LIN {X 0,Y 457.681,Z 997.987,A -85,B 0,C 180,E1 -8390.375,E2 -8390.375} C_VEL
LIN {X 0,Y 458.676,Z 987.154,A -85,B 0,C 180,E1 -8391.458,E2 -8391.458} C_VEL
LIN {X 0,Y 459.714,Z 975.478,A -85,B 0,C 180,E1 -8392.469,E2 -8392.469} C_VEL
LIN {X 0,Y 460.765,Z 963.447,A -85,B 0,C 180,E1 -8393.364,E2 -8393.364} C_VEL
LIN {X 0,Y 461.763,Z 951.373,A -85,B 0,C 180,E1 -8394.128,E2 -8394.128} C_VEL
LIN {X 0,Y 462.621,Z 938.572,A -85,B 0,C 180,E1 -8394.813,E2 -8394.813} C_VEL
LIN {X 0,Y 463.49,Z 925.141,A -85,B 0,C 180,E1 -8395.393,E2 -8395.393} C_VEL
LIN {X 0,Y 464.076,Z 912.216,A -85,B 0,C 180,E1 -8395.84,E2 -8395.84} C_VEL
LIN {X 0,Y 464.663,Z 898.95,A -85,B 0,C 180,E1 -8396.175,E2 -8396.175} C_VEL
LIN {X 0,Y 465.199,Z 876.109,A -85,B 0,C 180,E1 -8396.57,E2 -8396.57} C_VEL
LIN {X 0,Y 467.459,Z 725.355,A -85,B 0,C 180,E1 -8398.991,E2 -8398.991} C_VEL
LIN {X 0,Y 459.982,Z 695.02,A -85,B 0,C 180,E1 -8400.037,E2 -8400.037} C_VEL
LIN {X 0,Y 459.58,Z 692.84,A -85,B 0,C 180,E1 -8400.156,E2 -8400.156} C_VEL
LIN {X 0,Y 459.765,Z 687.054,A -85,B 0,C 180,E1 -8401.128,E2 -8401.128} C_VEL
LIN {X 0,Y 456.55,Z 673.441,A -85,B 0,C 180,E1 -8403.772,E2 -8403.772} C_VEL
LIN {X 0,Y 453.496,Z 662.065,A -85,B 0,C 180,E1 -8406.147,E2 -8406.147} C_VEL
LIN {X 0,Y 453.451,Z 661.817,A -85,B 0,C 180,E1 -8406.299,E2 -8406.299} C_VEL
LIN {X 0,Y 453.512,Z 661.81,A -85,B 0,C 180,E1 -8409.446,E2 -8409.446} C_VEL
LIN {X 0,Y 453.463,Z 661.814,A -85,B 0,C 180,E1 -8412.994,E2 -8412.994} C_VEL
LIN {X 0,Y 453.471,Z 661.808,A -85,B 0,C 180,E1 -8415.78,E2 -8415.78} C_VEL
LIN {X 0,Y 453.491,Z 661.792,A -85,B 0,C 180,E1 -8418.211,E2 -8418.211} C_VEL
LIN {X 0,Y 453.529,Z 661.801,A -85,B 0,C 180,E1 -8420.786,E2 -8420.786} C_VEL
LIN {X 0,Y 453.45,Z 661.794,A -85,B 0,C 180,E1 -8423.917,E2 -8423.917} C_VEL
LIN {X 0,Y 453.475,Z 661.808,A -85,B 0,C 180,E1 -8427.151,E2 -8427.151} C_VEL
LIN {X 0,Y 453.506,Z 661.775,A -85,B 0,C 180,E1 -8430.271,E2 -8430.271} C_VEL
LIN {X 0,Y 453.505,Z 661.795,A -85,B 0,C 180,E1 -8433.294,E2 -8433.294} C_VEL
LIN {X 0,Y 453.495,Z 661.808,A -85,B 0,C 180,E1 -8436.238,E2 -8436.238} C_VEL
LIN {X 0,Y 453.473,Z 661.809,A -85,B 0,C 180,E1 -8439.117,E2 -8439.117} C_VEL
LIN {X 0,Y 453.502,Z 661.798,A -85,B 0,C 180,E1 -8441.944,E2 -8441.944} C_VEL
LIN {X 0,Y 453.53,Z 661.807,A -85,B 0,C 180,E1 -8444.726,E2 -8444.726} C_VEL
LIN {X 0,Y 453.592,Z 661.788,A -85,B 0,C 180,E1 -8447.472,E2 -8447.472} C_VEL
LIN {X 0,Y 453.584,Z 661.788,A -85,B 0,C 180,E1 -8451.086,E2 -8451.086} C_VEL
LIN {X 0,Y 453.674,Z 661.781,A -85,B 0,C 180,E1 -8453.774,E2 -8453.774} C_VEL
LIN {X 0,Y 453.756,Z 661.766,A -85,B 0,C 180,E1 -8457.337,E2 -8457.337} C_VEL
LIN {X 0,Y 453.813,Z 661.765,A -85,B 0,C 180,E1 -8460,E2 -8460} C_VEL
LIN {X 0,Y 453.756,Z 661.76,A -85,B 0,C 180,E1 -8462.663,E2 -8462.663} C_VEL
LIN {X 0,Y 453.673,Z 661.78,A -85,B 0,C 180,E1 -8466.225,E2 -8466.225} C_VEL
LIN {X 0,Y 453.583,Z 661.789,A -85,B 0,C 180,E1 -8468.913,E2 -8468.913} C_VEL
LIN {X 0,Y 453.552,Z 661.786,A -85,B 0,C 180,E1 -8472.529,E2 -8472.529} C_VEL
LIN {X 0,Y 453.534,Z 661.799,A -85,B 0,C 180,E1 -8476.196,E2 -8476.196} C_VEL
LIN {X 0,Y 453.509,Z 661.801,A -85,B 0,C 180,E1 -8479.041,E2 -8479.041} C_VEL
LIN {X 0,Y 453.493,Z 661.804,A -85,B 0,C 180,E1 -8481.835,E2 -8481.835} C_VEL
LIN {X 0,Y 453.506,Z 661.806,A -85,B 0,C 180,E1 -8484.734,E2 -8484.734} C_VEL
LIN {X 0,Y 453.528,Z 661.776,A -85,B 0,C 180,E1 -8487.961,E2 -8487.961} C_VEL
LIN {X 0,Y 453.473,Z 661.798,A -85,B 0,C 180,E1 -8490.759,E2 -8490.759} C_VEL
LIN {X 0,Y 453.468,Z 661.806,A -85,B 0,C 180,E1 -8493.913,E2 -8493.913} C_VEL
LIN {X 0,Y 453.462,Z 661.792,A -85,B 0,C 180,E1 -8497.188,E2 -8497.188} C_VEL
LIN {X 0,Y 453.524,Z 661.804,A -85,B 0,C 180,E1 -8499.446,E2 -8499.446} C_VEL
LIN {X 0,Y 453.484,Z 661.813,A -85,B 0,C 180,E1 -8502.992,E2 -8502.992} C_VEL
LIN {X 0,Y 453.457,Z 661.812,A -85,B 0,C 180,E1 -8505.779,E2 -8505.779} C_VEL
LIN {X 0,Y 453.508,Z 661.81,A -85,B 0,C 180,E1 -8509.406,E2 -8509.406} C_VEL
LIN {X 0,Y 453.469,Z 661.81,A -85,B 0,C 180,E1 -8512.223,E2 -8512.223} C_VEL
LIN {X 0,Y 453.482,Z 661.811,A -85,B 0,C 180,E1 -8515.223,E2 -8515.223} C_VEL
LIN {X 0,Y 453.462,Z 661.811,A -85,B 0,C 180,E1 -8518.475,E2 -8518.475} C_VEL
LIN {X 0,Y 453.509,Z 661.806,A -85,B 0,C 180,E1 -8521.289,E2 -8521.289} C_VEL
LIN {X 0,Y 453.519,Z 661.808,A -85,B 0,C 180,E1 -8524.285,E2 -8524.285} C_VEL
LIN {X 0,Y 453.475,Z 661.81,A -85,B 0,C 180,E1 -8527.205,E2 -8527.205} C_VEL
LIN {X 0,Y 453.5,Z 661.811,A -85,B 0,C 180,E1 -8530.066,E2 -8530.066} C_VEL
LIN {X 0,Y 453.502,Z 661.807,A -85,B 0,C 180,E1 -8532.876,E2 -8532.876} C_VEL
LIN {X 0,Y 453.509,Z 661.807,A -85,B 0,C 180,E1 -8535.644,E2 -8535.644} C_VEL
LIN {X 0,Y 453.556,Z 661.803,A -85,B 0,C 180,E1 -8538.379,E2 -8538.379} C_VEL
LIN {X 0,Y 453.648,Z 661.789,A -85,B 0,C 180,E1 -8541.985,E2 -8541.985} C_VEL
LIN {X 0,Y 453.633,Z 661.791,A -85,B 0,C 180,E1 -8543.096,E2 -8543.096} C_VEL
LIN {X 0,Y 452.948,Z 661.876,A -85,B 0,C 180,E1 -8543.836,E2 -8543.836} C_VEL
LIN {X 0,Y 450,Z 662.245,A -85,B 0,C 180,E1 -8545.038,E2 -8545.038} C_VEL
LIN {X 0,Y 447.578,Z 662.546,A -85,B 0,C 180,E1 -8546.007,E2 -8546.007} C_VEL
LIN {X 0,Y 446.641,Z 662.663,A -85,B 0,C 180,E1 -8546.758,E2 -8546.758} C_VEL
LIN {X 0,Y 446.621,Z 662.665,A -85,B 0,C 180,E1 -8547.011,E2 -8547.011} C_VEL
LIN {X 0,Y 446.79,Z 662.644,A -85,B 0,C 180,E1 -8550,E2 -8550} C_VEL
LIN {X 0,Y 446.706,Z 662.656,A -85,B 0,C 180,E1 -8552.705,E2 -8552.705} C_VEL
LIN {X 0,Y 446.643,Z 662.661,A -85,B 0,C 180,E1 -8556.324,E2 -8556.324} C_VEL
LIN {X 0,Y 446.534,Z 662.676,A -85,B 0,C 180,E1 -8559.055,E2 -8559.055} C_VEL
LIN {X 0,Y 446.517,Z 662.676,A -85,B 0,C 180,E1 -8562.729,E2 -8562.729} C_VEL
LIN {X 0,Y 446.492,Z 662.68,A -85,B 0,C 180,E1 -8566.228,E2 -8566.228} C_VEL
LIN {X 0,Y 446.464,Z 662.684,A -85,B 0,C 180,E1 -8569.303,E2 -8569.303} C_VEL
LIN {X 0,Y 446.414,Z 662.692,A -85,B 0,C 180,E1 -8572.199,E2 -8572.199} C_VEL
LIN {X 0,Y 446.452,Z 662.685,A -85,B 0,C 180,E1 -8575.152,E2 -8575.152} C_VEL
LIN {X 0,Y 446.479,Z 662.685,A -85,B 0,C 180,E1 -8578.178,E2 -8578.178} C_VEL
LIN {X 0,Y 446.413,Z 662.689,A -85,B 0,C 180,E1 -8581.3,E2 -8581.3} C_VEL
LIN {X 0,Y 446.424,Z 662.691,A -85,B 0,C 180,E1 -8584.522,E2 -8584.522} C_VEL
LIN {X 0,Y 446.429,Z 662.69,A -85,B 0,C 180,E1 -8588.082,E2 -8588.082} C_VEL
LIN {X 0,Y 446.435,Z 662.689,A -85,B 0,C 180,E1 -8590.92,E2 -8590.92} C_VEL
LIN {X 0,Y 446.393,Z 662.691,A -85,B 0,C 180,E1 -8593.845,E2 -8593.845} C_VEL
LIN {X 0,Y 446.438,Z 662.688,A -85,B 0,C 180,E1 -8596.396,E2 -8596.396} C_VEL
LIN {X 0,Y 446.46,Z 662.682,A -85,B 0,C 180,E1 -8599.805,E2 -8599.805} C_VEL
LIN {X 0,Y 446.425,Z 662.68,A -85,B 0,C 180,E1 -8602.123,E2 -8602.123} C_VEL
LIN {X 0,Y 446.421,Z 662.675,A -85,B 0,C 180,E1 -8605.477,E2 -8605.477} C_VEL
LIN {X 0,Y 446.41,Z 662.687,A -85,B 0,C 180,E1 -8608.7,E2 -8608.7} C_VEL
LIN {X 0,Y 446.474,Z 662.651,A -85,B 0,C 180,E1 -8611.821,E2 -8611.821} C_VEL
LIN {X 0,Y 446.449,Z 662.682,A -85,B 0,C 180,E1 -8614.848,E2 -8614.848} C_VEL
LIN {X 0,Y 446.474,Z 662.678,A -85,B 0,C 180,E1 -8618.233,E2 -8618.233} C_VEL
LIN {X 0,Y 446.446,Z 662.68,A -85,B 0,C 180,E1 -8621.649,E2 -8621.649} C_VEL
LIN {X 0,Y 446.496,Z 662.678,A -85,B 0,C 180,E1 -8624.48,E2 -8624.48} C_VEL
LIN {X 0,Y 446.508,Z 662.671,A -85,B 0,C 180,E1 -8628.193,E2 -8628.193} C_VEL
LIN {X 0,Y 446.589,Z 662.659,A -85,B 0,C 180,E1 -8631.858,E2 -8631.858} C_VEL
LIN {X 0,Y 446.643,Z 662.663,A -85,B 0,C 180,E1 -8634.583,E2 -8634.583} C_VEL
LIN {X 0,Y 446.7,Z 662.639,A -85,B 0,C 180,E1 -8637.295,E2 -8637.295} C_VEL
LIN {X 0,Y 446.784,Z 662.641,A -85,B 0,C 180,E1 -8640,E2 -8640} C_VEL
LIN {X 0,Y 446.7,Z 662.645,A -85,B 0,C 180,E1 -8642.706,E2 -8642.706} C_VEL
LIN {X 0,Y 446.642,Z 662.658,A -85,B 0,C 180,E1 -8646.324,E2 -8646.324} C_VEL
LIN {X 0,Y 446.53,Z 662.668,A -85,B 0,C 180,E1 -8649.056,E2 -8649.056} C_VEL
LIN {X 0,Y 446.524,Z 662.667,A -85,B 0,C 180,E1 -8652.73,E2 -8652.73} C_VEL
LIN {X 0,Y 446.48,Z 662.676,A -85,B 0,C 180,E1 -8656.46,E2 -8656.46} C_VEL
LIN {X 0,Y 446.46,Z 662.681,A -85,B 0,C 180,E1 -8659.304,E2 -8659.304} C_VEL
LIN {X 0,Y 446.409,Z 662.679,A -85,B 0,C 180,E1 -8662.2,E2 -8662.2} C_VEL
LIN {X 0,Y 446.45,Z 662.685,A -85,B 0,C 180,E1 -8665.153,E2 -8665.153} C_VEL
LIN {X 0,Y 446.476,Z 662.645,A -85,B 0,C 180,E1 -8668.179,E2 -8668.179} C_VEL
LIN {X 0,Y 446.412,Z 662.681,A -85,B 0,C 180,E1 -8671.301,E2 -8671.301} C_VEL
LIN {X 0,Y 446.423,Z 662.674,A -85,B 0,C 180,E1 -8674.524,E2 -8674.524} C_VEL
LIN {X 0,Y 446.433,Z 662.687,A -85,B 0,C 180,E1 -8678.084,E2 -8678.084} C_VEL
LIN {X 0,Y 446.441,Z 662.667,A -85,B 0,C 180,E1 -8680.921,E2 -8680.921} C_VEL
LIN {X 0,Y 446.439,Z 662.688,A -85,B 0,C 180,E1 -8683.841,E2 -8683.841} C_VEL
LIN {X 0,Y 446.415,Z 662.68,A -85,B 0,C 180,E1 -8686.401,E2 -8686.401} C_VEL
LIN {X 0,Y 446.446,Z 662.68,A -85,B 0,C 180,E1 -8689.804,E2 -8689.804} C_VEL
LIN {X 0,Y 446.405,Z 662.659,A -85,B 0,C 180,E1 -8692.122,E2 -8692.122} C_VEL
LIN {X 0,Y 446.413,Z 662.764,A -85,B 0,C 180,E1 -8693.315,E2 -8693.315} C_VEL
LIN {X 0,Y 446.806,Z 664.307,A -85,B 0,C 180,E1 -8693.72,E2 -8693.72} C_VEL
LIN {X 0,Y 450.168,Z 677.011,A -85,B 0,C 180,E1 -8696.383,E2 -8696.383} C_VEL
LIN {X 0,Y 453.035,Z 689.272,A -85,B 0,C 180,E1 -8698.796,E2 -8698.796} C_VEL
LIN {X 0,Y 452.916,Z 692.897,A -85,B 0,C 180,E1 -8699.386,E2 -8699.386} C_VEL
LIN {X 0,Y 460.04,Z 721.732,A -85,B 0,C 180,E1 -8700.437,E2 -8700.437} C_VEL
LIN {X 0,Y 461.227,Z 726.758,A -85,B 0,C 180,E1 -8700.607,E2 -8700.607} C_VEL
LIN {X 0,Y 458.465,Z 895.176,A -85,B 0,C 180,E1 -8703.365,E2 -8703.365} C_VEL
LIN {X 0,Y 457.913,Z 908.094,A -85,B 0,C 180,E1 -8703.664,E2 -8703.664} C_VEL
LIN {X 0,Y 457.288,Z 920.455,A -85,B 0,C 180,E1 -8704.054,E2 -8704.054} C_VEL
LIN {X 0,Y 456.509,Z 933.579,A -85,B 0,C 180,E1 -8704.588,E2 -8704.588} C_VEL
LIN {X 0,Y 455.674,Z 944.969,A -85,B 0,C 180,E1 -8705.148,E2 -8705.148} C_VEL
LIN {X 0,Y 454.721,Z 957.622,A -85,B 0,C 180,E1 -8705.901,E2 -8705.901} C_VEL
LIN {X 0,Y 453.634,Z 969.515,A -85,B 0,C 180,E1 -8706.731,E2 -8706.731} C_VEL
LIN {X 0,Y 452.493,Z 981.957,A -85,B 0,C 180,E1 -8707.754,E2 -8707.754} C_VEL
LIN {X 0,Y 451.423,Z 992.762,A -85,B 0,C 180,E1 -8708.779,E2 -8708.779} C_VEL
LIN {X 0,Y 450.318,Z 1003.265,A -85,B 0,C 180,E1 -8709.92,E2 -8709.92} C_VEL
LIN {X 0,Y 449.455,Z 1012.541,A -85,B 0,C 180,E1 -8711.068,E2 -8711.068} C_VEL
LIN {X 0,Y 448.523,Z 1022.278,A -85,B 0,C 180,E1 -8712.445,E2 -8712.445} C_VEL
LIN {X 0,Y 447.768,Z 1030.805,A -85,B 0,C 180,E1 -8713.824,E2 -8713.824} C_VEL
LIN {X 0,Y 446.987,Z 1039.406,A -85,B 0,C 180,E1 -8715.43,E2 -8715.43} C_VEL
LIN {X 0,Y 446.528,Z 1045.836,A -85,B 0,C 180,E1 -8716.808,E2 -8716.808} C_VEL
LIN {X 0,Y 446.169,Z 1051.474,A -85,B 0,C 180,E1 -8718.184,E2 -8718.184} C_VEL
LIN {X 0,Y 445.72,Z 1057.738,A -85,B 0,C 180,E1 -8720.012,E2 -8720.012} C_VEL
LIN {X 0,Y 445.567,Z 1062.829,A -85,B 0,C 180,E1 -8721.839,E2 -8721.839} C_VEL
LIN {X 0,Y 445.487,Z 1066.82,A -85,B 0,C 180,E1 -8723.66,E2 -8723.66} C_VEL
LIN {X 0,Y 445.363,Z 1069.763,A -85,B 0,C 180,E1 -8725.475,E2 -8725.475} C_VEL
LIN {X 0,Y 445.332,Z 1070.944,A -85,B 0,C 180,E1 -8726.381,E2 -8726.381} C_VEL
LIN {X 0,Y 445.346,Z 1072.406,A -85,B 0,C 180,E1 -8728.191,E2 -8728.191} C_VEL
LIN {X 0,Y 445.338,Z 1072.89,A -85,B 0,C 180,E1 -8730,E2 -8730} C_VEL
LIN {X 0,Y 445.346,Z 1072.406,A -85,B 0,C 180,E1 -8731.809,E2 -8731.809} C_VEL
LIN {X 0,Y 445.332,Z 1070.944,A -85,B 0,C 180,E1 -8733.619,E2 -8733.619} C_VEL
LIN {X 0,Y 445.403,Z 1068.487,A -85,B 0,C 180,E1 -8735.432,E2 -8735.432} C_VEL
LIN {X 0,Y 445.538,Z 1063.916,A -85,B 0,C 180,E1 -8737.705,E2 -8737.705} C_VEL
LIN {X 0,Y 445.632,Z 1060.432,A -85,B 0,C 180,E1 -8739.074,E2 -8739.074} C_VEL
LIN {X 0,Y 445.939,Z 1054.714,A -85,B 0,C 180,E1 -8740.901,E2 -8740.901} C_VEL
LIN {X 0,Y 446.336,Z 1048.664,A -85,B 0,C 180,E1 -8742.513,E2 -8742.513} C_VEL
LIN {X 0,Y 446.796,Z 1041.627,A -85,B 0,C 180,E1 -8744.111,E2 -8744.111} C_VEL
LIN {X 0,Y 447.422,Z 1034.645,A -85,B 0,C 180,E1 -8745.487,E2 -8745.487} C_VEL
LIN {X 0,Y 448.159,Z 1026.186,A -85,B 0,C 180,E1 -8746.943,E2 -8746.943} C_VEL
LIN {X 0,Y 448.963,Z 1017.559,A -85,B 0,C 180,E1 -8748.244,E2 -8748.244} C_VEL
LIN {X 0,Y 449.782,Z 1008.987,A -85,B 0,C 180,E1 -8749.392,E2 -8749.392} C_VEL
LIN {X 0,Y 450.846,Z 998.67,A -85,B 0,C 180,E1 -8750.6,E2 -8750.6} C_VEL
LIN {X 0,Y 451.991,Z 986.946,A -85,B 0,C 180,E1 -8751.791,E2 -8751.791} C_VEL
LIN {X 0,Y 453.089,Z 975.27,A -85,B 0,C 180,E1 -8752.816,E2 -8752.816} C_VEL
LIN {X 0,Y 454.194,Z 963.24,A -85,B 0,C 180,E1 -8753.722,E2 -8753.722} C_VEL
LIN {X 0,Y 455.295,Z 950.188,A -85,B 0,C 180,E1 -8754.554,E2 -8754.554} C_VEL
LIN {X 0,Y 456.156,Z 938.366,A -85,B 0,C 180,E1 -8755.189,E2 -8755.189} C_VEL
LIN {X 0,Y 457.071,Z 924.935,A -85,B 0,C 180,E1 -8755.775,E2 -8755.775} C_VEL
LIN {X 0,Y 457.701,Z 912.011,A -85,B 0,C 180,E1 -8756.227,E2 -8756.227} C_VEL
LIN {X 0,Y 458.358,Z 897.828,A -85,B 0,C 180,E1 -8756.583,E2 -8756.583} C_VEL
LIN {X 0,Y 458.955,Z 869.586,A -85,B 0,C 180,E1 -8757.069,E2 -8757.069} C_VEL
LIN {X 0,Y 461.266,Z 726.901,A -85,B 0,C 180,E1 -8759.387,E2 -8759.387} C_VEL
LIN {X 0,Y 453.396,Z 694.842,A -85,B 0,C 180,E1 -8760.519,E2 -8760.519} C_VEL
LIN {X 0,Y 452.958,Z 692.786,A -85,B 0,C 180,E1 -8760.62,E2 -8760.62} C_VEL
LIN {X 0,Y 453.046,Z 689.286,A -85,B 0,C 180,E1 -8761.201,E2 -8761.201} C_VEL
LIN {X 0,Y 449.639,Z 674.79,A -85,B 0,C 180,E1 -8764.065,E2 -8764.065} C_VEL
LIN {X 0,Y 446.433,Z 662.959,A -85,B 0,C 180,E1 -8766.595,E2 -8766.595} C_VEL
LIN {X 0,Y 446.398,Z 662.695,A -85,B 0,C 180,E1 -8766.745,E2 -8766.745} C_VEL
LIN {X 0,Y 446.473,Z 662.685,A -85,B 0,C 180,E1 -8769.528,E2 -8769.528} C_VEL
LIN {X 0,Y 446.427,Z 662.688,A -85,B 0,C 180,E1 -8772.603,E2 -8772.603} C_VEL
LIN {X 0,Y 446.452,Z 662.671,A -85,B 0,C 180,E1 -8775.102,E2 -8775.102} C_VEL
LIN {X 0,Y 446.438,Z 662.667,A -85,B 0,C 180,E1 -8778.61,E2 -8778.61} C_VEL
LIN {X 0,Y 446.471,Z 662.68,A -85,B 0,C 180,E1 -8780.976,E2 -8780.976} C_VEL
LIN {X 0,Y 446.414,Z 662.668,A -85,B 0,C 180,E1 -8784.373,E2 -8784.373} C_VEL
LIN {X 0,Y 446.415,Z 662.69,A -85,B 0,C 180,E1 -8787.638,E2 -8787.638} C_VEL
LIN {X 0,Y 446.461,Z 662.646,A -85,B 0,C 180,E1 -8790.791,E2 -8790.791} C_VEL
LIN {X 0,Y 446.469,Z 662.674,A -85,B 0,C 180,E1 -8793.848,E2 -8793.848} C_VEL
LIN {X 0,Y 446.42,Z 662.68,A -85,B 0,C 180,E1 -8796.823,E2 -8796.823} C_VEL
LIN {X 0,Y 446.435,Z 662.685,A -85,B 0,C 180,E1 -8799.737,E2 -8799.737} C_VEL
LIN {X 0,Y 446.454,Z 662.677,A -85,B 0,C 180,E1 -8802.597,E2 -8802.597} C_VEL
LIN {X 0,Y 446.462,Z 662.679,A -85,B 0,C 180,E1 -8805.412,E2 -8805.412} C_VEL
LIN {X 0,Y 446.537,Z 662.666,A -85,B 0,C 180,E1 -8808.193,E2 -8808.193} C_VEL
LIN {X 0,Y 446.59,Z 662.652,A -85,B 0,C 180,E1 -8811.857,E2 -8811.857} C_VEL
LIN {X 0,Y 446.643,Z 662.658,A -85,B 0,C 180,E1 -8814.582,E2 -8814.582} C_VEL
LIN {X 0,Y 446.7,Z 662.644,A -85,B 0,C 180,E1 -8817.294,E2 -8817.294} C_VEL
LIN {X 0,Y 446.784,Z 662.641,A -85,B 0,C 180,E1 -8820,E2 -8820} C_VEL
LIN {X 0,Y 446.7,Z 662.638,A -85,B 0,C 180,E1 -8822.705,E2 -8822.705} C_VEL
LIN {X 0,Y 446.641,Z 662.655,A -85,B 0,C 180,E1 -8826.323,E2 -8826.323} C_VEL
LIN {X 0,Y 446.528,Z 662.668,A -85,B 0,C 180,E1 -8829.055,E2 -8829.055} C_VEL
LIN {X 0,Y 446.51,Z 662.662,A -85,B 0,C 180,E1 -8832.73,E2 -8832.73} C_VEL
LIN {X 0,Y 446.485,Z 662.677,A -85,B 0,C 180,E1 -8836.228,E2 -8836.228} C_VEL
LIN {X 0,Y 446.46,Z 662.679,A -85,B 0,C 180,E1 -8839.303,E2 -8839.303} C_VEL
LIN {X 0,Y 446.43,Z 662.681,A -85,B 0,C 180,E1 -8842.199,E2 -8842.199} C_VEL
LIN {X 0,Y 446.449,Z 662.682,A -85,B 0,C 180,E1 -8845.152,E2 -8845.152} C_VEL
LIN {X 0,Y 446.474,Z 662.651,A -85,B 0,C 180,E1 -8848.179,E2 -8848.179} C_VEL
LIN {X 0,Y 446.41,Z 662.687,A -85,B 0,C 180,E1 -8851.3,E2 -8851.3} C_VEL
LIN {X 0,Y 446.421,Z 662.675,A -85,B 0,C 180,E1 -8854.523,E2 -8854.523} C_VEL
LIN {X 0,Y 446.429,Z 662.68,A -85,B 0,C 180,E1 -8858.083,E2 -8858.083} C_VEL
LIN {X 0,Y 446.439,Z 662.69,A -85,B 0,C 180,E1 -8860.921,E2 -8860.921} C_VEL
LIN {X 0,Y 446.437,Z 662.686,A -85,B 0,C 180,E1 -8863.841,E2 -8863.841} C_VEL
LIN {X 0,Y 446.391,Z 662.691,A -85,B 0,C 180,E1 -8866.404,E2 -8866.404} C_VEL
LIN {X 0,Y 446.46,Z 662.684,A -85,B 0,C 180,E1 -8869.805,E2 -8869.805} C_VEL
LIN {X 0,Y 446.425,Z 662.688,A -85,B 0,C 180,E1 -8872.124,E2 -8872.124} C_VEL
LIN {X 0,Y 446.424,Z 662.691,A -85,B 0,C 180,E1 -8875.478,E2 -8875.478} C_VEL
LIN {X 0,Y 446.413,Z 662.689,A -85,B 0,C 180,E1 -8878.7,E2 -8878.7} C_VEL
LIN {X 0,Y 446.479,Z 662.685,A -85,B 0,C 180,E1 -8881.822,E2 -8881.822} C_VEL
LIN {X 0,Y 446.452,Z 662.685,A -85,B 0,C 180,E1 -8884.848,E2 -8884.848} C_VEL
LIN {X 0,Y 446.443,Z 662.688,A -85,B 0,C 180,E1 -8888.245,E2 -8888.245} C_VEL
LIN {X 0,Y 446.453,Z 662.687,A -85,B 0,C 180,E1 -8891.65,E2 -8891.65} C_VEL
LIN {X 0,Y 446.503,Z 662.68,A -85,B 0,C 180,E1 -8894.48,E2 -8894.48} C_VEL
LIN {X 0,Y 446.513,Z 662.681,A -85,B 0,C 180,E1 -8898.193,E2 -8898.193} C_VEL
LIN {X 0,Y 446.596,Z 662.667,A -85,B 0,C 180,E1 -8901.858,E2 -8901.858} C_VEL
LIN {X 0,Y 446.642,Z 662.664,A -85,B 0,C 180,E1 -8904.583,E2 -8904.583} C_VEL
LIN {X 0,Y 446.621,Z 662.665,A -85,B 0,C 180,E1 -8907.011,E2 -8907.011} C_VEL
LIN {X 0,Y 446.104,Z 662.732,A -85,B 0,C 180,E1 -8907.764,E2 -8907.764} C_VEL
LIN {X 0,Y 443.287,Z 663.087,A -85,B 0,C 180,E1 -8908.987,E2 -8908.987} C_VEL
LIN {X 0,Y 440.8,Z 663.396,A -85,B 0,C 180,E1 -8909.974,E2 -8909.974} C_VEL
LIN {X 0,Y 439.711,Z 663.528,A -85,B 0,C 180,E1 -8910.737,E2 -8910.737} C_VEL
LIN {X 0,Y 439.618,Z 663.537,A -85,B 0,C 180,E1 -8910.996,E2 -8910.996} C_VEL
LIN {X 0,Y 439.652,Z 663.535,A -85,B 0,C 180,E1 -8912.749,E2 -8912.749} C_VEL
LIN {X 0,Y 439.615,Z 663.537,A -85,B 0,C 180,E1 -8916.425,E2 -8916.425} C_VEL
LIN {X 0,Y 439.496,Z 663.554,A -85,B 0,C 180,E1 -8919.201,E2 -8919.201} C_VEL
LIN {X 0,Y 439.461,Z 663.556,A -85,B 0,C 180,E1 -8922.937,E2 -8922.937} C_VEL
LIN {X 0,Y 439.443,Z 663.557,A -85,B 0,C 180,E1 -8926.349,E2 -8926.349} C_VEL
LIN {X 0,Y 439.398,Z 663.565,A -85,B 0,C 180,E1 -8929.626,E2 -8929.626} C_VEL
LIN {X 0,Y 439.36,Z 663.57,A -85,B 0,C 180,E1 -8932.575,E2 -8932.575} C_VEL
LIN {X 0,Y 439.4,Z 663.566,A -85,B 0,C 180,E1 -8935.584,E2 -8935.584} C_VEL
LIN {X 0,Y 439.419,Z 663.562,A -85,B 0,C 180,E1 -8938.672,E2 -8938.672} C_VEL
LIN {X 0,Y 439.368,Z 663.568,A -85,B 0,C 180,E1 -8941.86,E2 -8941.86} C_VEL
LIN {X 0,Y 439.394,Z 663.564,A -85,B 0,C 180,E1 -8945.155,E2 -8945.155} C_VEL
LIN {X 0,Y 439.39,Z 663.567,A -85,B 0,C 180,E1 -8948.593,E2 -8948.593} C_VEL
LIN {X 0,Y 439.39,Z 663.565,A -85,B 0,C 180,E1 -8951.258,E2 -8951.258} C_VEL
LIN {X 0,Y 439.394,Z 663.568,A -85,B 0,C 180,E1 -8954.729,E2 -8954.729} C_VEL
LIN {X 0,Y 439.404,Z 663.562,A -85,B 0,C 180,E1 -8957.797,E2 -8957.797} C_VEL
LIN {X 0,Y 439.443,Z 663.557,A -85,B 0,C 180,E1 -8960.23,E2 -8960.23} C_VEL
LIN {X 0,Y 439.368,Z 663.536,A -85,B 0,C 180,E1 -8963.713,E2 -8963.713} C_VEL
LIN {X 0,Y 439.363,Z 663.568,A -85,B 0,C 180,E1 -8967.054,E2 -8967.054} C_VEL
LIN {X 0,Y 439.386,Z 663.538,A -85,B 0,C 180,E1 -8970.275,E2 -8970.275} C_VEL
LIN {X 0,Y 439.42,Z 663.545,A -85,B 0,C 180,E1 -8973.396,E2 -8973.396} C_VEL
LIN {X 0,Y 439.383,Z 663.56,A -85,B 0,C 180,E1 -8976.43,E2 -8976.43} C_VEL
LIN {X 0,Y 439.403,Z 663.56,A -85,B 0,C 180,E1 -8979.398,E2 -8979.398} C_VEL
LIN {X 0,Y 439.42,Z 663.551,A -85,B 0,C 180,E1 -8982.309,E2 -8982.309} C_VEL
LIN {X 0,Y 439.437,Z 663.555,A -85,B 0,C 180,E1 -8985.174,E2 -8985.174} C_VEL
LIN {X 0,Y 439.474,Z 663.543,A -85,B 0,C 180,E1 -8988.001,E2 -8988.001} C_VEL
LIN {X 0,Y 439.537,Z 663.538,A -85,B 0,C 180,E1 -8991.726,E2 -8991.726} C_VEL
LIN {X 0,Y 439.618,Z 663.539,A -85,B 0,C 180,E1 -8994.496,E2 -8994.496} C_VEL
LIN {X 0,Y 439.626,Z 663.523,A -85,B 0,C 180,E1 -8998.168,E2 -8998.168} C_VEL
LIN {X 0,Y 439.754,Z 663.517,A -85,B 0,C 180,E1 -9000,E2 -9000} C_VEL
LIN {X 0,Y 439.647,Z 663.523,A -85,B 0,C 180,E1 -9002.749,E2 -9002.749} C_VEL
LIN {X 0,Y 439.612,Z 663.535,A -85,B 0,C 180,E1 -9006.425,E2 -9006.425} C_VEL
LIN {X 0,Y 439.492,Z 663.547,A -85,B 0,C 180,E1 -9009.202,E2 -9009.202} C_VEL
LIN {X 0,Y 439.495,Z 663.542,A -85,B 0,C 180,E1 -9012.727,E2 -9012.727} C_VEL
LIN {X 0,Y 439.438,Z 663.553,A -85,B 0,C 180,E1 -9016.349,E2 -9016.349} C_VEL
LIN {X 0,Y 439.422,Z 663.564,A -85,B 0,C 180,E1 -9019.625,E2 -9019.625} C_VEL
LIN {X 0,Y 439.356,Z 663.556,A -85,B 0,C 180,E1 -9022.576,E2 -9022.576} C_VEL
LIN {X 0,Y 439.397,Z 663.562,A -85,B 0,C 180,E1 -9025.585,E2 -9025.585} C_VEL
LIN {X 0,Y 439.417,Z 663.52,A -85,B 0,C 180,E1 -9028.674,E2 -9028.674} C_VEL
LIN {X 0,Y 439.367,Z 663.565,A -85,B 0,C 180,E1 -9031.861,E2 -9031.861} C_VEL
LIN {X 0,Y 439.393,Z 663.545,A -85,B 0,C 180,E1 -9035.157,E2 -9035.157} C_VEL
LIN {X 0,Y 439.394,Z 663.565,A -85,B 0,C 180,E1 -9038.594,E2 -9038.594} C_VEL
LIN {X 0,Y 439.399,Z 663.543,A -85,B 0,C 180,E1 -9041.26,E2 -9041.26} C_VEL
LIN {X 0,Y 439.404,Z 663.551,A -85,B 0,C 180,E1 -9044.729,E2 -9044.729} C_VEL
LIN {X 0,Y 439.393,Z 663.565,A -85,B 0,C 180,E1 -9047.797,E2 -9047.797} C_VEL
LIN {X 0,Y 439.432,Z 663.56,A -85,B 0,C 180,E1 -9050.229,E2 -9050.229} C_VEL
LIN {X 0,Y 439.376,Z 663.703,A -85,B 0,C 180,E1 -9052.881,E2 -9052.881} C_VEL
LIN {X 0,Y 441.412,Z 671.184,A -85,B 0,C 180,E1 -9054.575,E2 -9054.575} C_VEL
LIN {X 0,Y 444.555,Z 683.682,A -85,B 0,C 180,E1 -9057.171,E2 -9057.171} C_VEL
LIN {X 0,Y 446.293,Z 691.825,A -85,B 0,C 180,E1 -9058.77,E2 -9058.77} C_VEL
LIN {X 0,Y 446.398,Z 693.117,A -85,B 0,C 180,E1 -9058.913,E2 -9058.913} C_VEL
LIN {X 0,Y 453.553,Z 721.825,A -85,B 0,C 180,E1 -9059.976,E2 -9059.976} C_VEL
LIN {X 0,Y 455.048,Z 728.255,A -85,B 0,C 180,E1 -9060.198,E2 -9060.198} C_VEL
LIN {X 0,Y 452.13,Z 895.322,A -85,B 0,C 180,E1 -9062.97,E2 -9062.97} C_VEL
LIN {X 0,Y 451.568,Z 907.889,A -85,B 0,C 180,E1 -9063.265,E2 -9063.265} C_VEL
LIN {X 0,Y 450.914,Z 919.502,A -85,B 0,C 180,E1 -9063.628,E2 -9063.628} C_VEL
LIN {X 0,Y 450.088,Z 933.373,A -85,B 0,C 180,E1 -9064.199,E2 -9064.199} C_VEL
LIN {X 0,Y 449.191,Z 944.761,A -85,B 0,C 180,E1 -9064.765,E2 -9064.765} C_VEL
LIN {X 0,Y 448.108,Z 958.364,A -85,B 0,C 180,E1 -9065.592,E2 -9065.592} C_VEL
LIN {X 0,Y 446.913,Z 970.747,A -85,B 0,C 180,E1 -9066.483,E2 -9066.483} C_VEL
LIN {X 0,Y 445.875,Z 981.75,A -85,B 0,C 180,E1 -9067.406,E2 -9067.406} C_VEL
LIN {X 0,Y 444.719,Z 992.554,A -85,B 0,C 180,E1 -9068.444,E2 -9068.444} C_VEL
LIN {X 0,Y 443.571,Z 1003.056,A -85,B 0,C 180,E1 -9069.601,E2 -9069.601} C_VEL
LIN {X 0,Y 442.665,Z 1012.333,A -85,B 0,C 180,E1 -9070.766,E2 -9070.766} C_VEL
LIN {X 0,Y 441.629,Z 1022.068,A -85,B 0,C 180,E1 -9072.162,E2 -9072.162} C_VEL
LIN {X 0,Y 440.846,Z 1030.597,A -85,B 0,C 180,E1 -9073.563,E2 -9073.563} C_VEL
LIN {X 0,Y 439.993,Z 1039.196,A -85,B 0,C 180,E1 -9075.193,E2 -9075.193} C_VEL
LIN {X 0,Y 439.515,Z 1045.628,A -85,B 0,C 180,E1 -9076.594,E2 -9076.594} C_VEL
LIN {X 0,Y 438.983,Z 1052.885,A -85,B 0,C 180,E1 -9078.456,E2 -9078.456} C_VEL
LIN {X 0,Y 438.662,Z 1057.531,A -85,B 0,C 180,E1 -9079.85,E2 -9079.85} C_VEL
LIN {X 0,Y 438.475,Z 1062.622,A -85,B 0,C 180,E1 -9081.706,E2 -9081.706} C_VEL
LIN {X 0,Y 438.393,Z 1066.848,A -85,B 0,C 180,E1 -9083.687,E2 -9083.687} C_VEL
LIN {X 0,Y 438.286,Z 1069.558,A -85,B 0,C 180,E1 -9085.401,E2 -9085.401} C_VEL
LIN {X 0,Y 438.235,Z 1070.738,A -85,B 0,C 180,E1 -9086.322,E2 -9086.322} C_VEL
LIN {X 0,Y 438.268,Z 1072.201,A -85,B 0,C 180,E1 -9088.162,E2 -9088.162} C_VEL
LIN {X 0,Y 438.249,Z 1072.685,A -85,B 0,C 180,E1 -9090,E2 -9090} C_VEL
LIN {X 0,Y 438.268,Z 1072.201,A -85,B 0,C 180,E1 -9091.838,E2 -9091.838} C_VEL
LIN {X 0,Y 438.235,Z 1070.738,A -85,B 0,C 180,E1 -9093.678,E2 -9093.678} C_VEL
LIN {X 0,Y 438.311,Z 1068.281,A -85,B 0,C 180,E1 -9095.521,E2 -9095.521} C_VEL
LIN {X 0,Y 438.462,Z 1063.709,A -85,B 0,C 180,E1 -9097.83,E2 -9097.83} C_VEL
LIN {X 0,Y 438.565,Z 1060.225,A -85,B 0,C 180,E1 -9099.221,E2 -9099.221} C_VEL
LIN {X 0,Y 438.898,Z 1054.506,A -85,B 0,C 180,E1 -9101.078,E2 -9101.078} C_VEL
LIN {X 0,Y 439.265,Z 1048.985,A -85,B 0,C 180,E1 -9102.588,E2 -9102.588} C_VEL
LIN {X 0,Y 439.808,Z 1041.419,A -85,B 0,C 180,E1 -9104.34,E2 -9104.34} C_VEL
LIN {X 0,Y 440.506,Z 1034.438,A -85,B 0,C 180,E1 -9105.737,E2 -9105.737} C_VEL
LIN {X 0,Y 441.207,Z 1026.638,A -85,B 0,C 180,E1 -9107.11,E2 -9107.11} C_VEL
LIN {X 0,Y 442.094,Z 1017.35,A -85,B 0,C 180,E1 -9108.538,E2 -9108.538} C_VEL
LIN {X 0,Y 442.986,Z 1008.778,A -85,B 0,C 180,E1 -9109.702,E2 -9109.702} C_VEL
LIN {X 0,Y 444.232,Z 997.512,A -85,B 0,C 180,E1 -9111.027,E2 -9111.027} C_VEL
LIN {X 0,Y 445.323,Z 986.738,A -85,B 0,C 180,E1 -9112.134,E2 -9112.134} C_VEL
LIN {X 0,Y 446.444,Z 975.061,A -85,B 0,C 180,E1 -9113.175,E2 -9113.175} C_VEL
LIN {X 0,Y 447.652,Z 963.033,A -85,B 0,C 180,E1 -9114.091,E2 -9114.091} C_VEL
LIN {X 0,Y 448.778,Z 950.121,A -85,B 0,C 180,E1 -9114.925,E2 -9114.925} C_VEL
LIN {X 0,Y 449.735,Z 938.16,A -85,B 0,C 180,E1 -9115.574,E2 -9115.574} C_VEL
LIN {X 0,Y 450.679,Z 924.729,A -85,B 0,C 180,E1 -9116.169,E2 -9116.169} C_VEL
LIN {X 0,Y 451.329,Z 911.805,A -85,B 0,C 180,E1 -9116.626,E2 -9116.626} C_VEL
LIN {X 0,Y 452.013,Z 897.842,A -85,B 0,C 180,E1 -9116.982,E2 -9116.982} C_VEL
LIN {X 0,Y 452.606,Z 870.46,A -85,B 0,C 180,E1 -9117.462,E2 -9117.462} C_VEL
LIN {X 0,Y 455.051,Z 728.321,A -85,B 0,C 180,E1 -9119.8,E2 -9119.8} C_VEL
LIN {X 0,Y 447.971,Z 699.056,A -85,B 0,C 180,E1 -9120.849,E2 -9120.849} C_VEL
LIN {X 0,Y 446.342,Z 692.486,A -85,B 0,C 180,E1 -9121.13,E2 -9121.13} C_VEL
LIN {X 0,Y 445.579,Z 687.975,A -85,B 0,C 180,E1 -9121.97,E2 -9121.97} C_VEL
LIN {X 0,Y 442.085,Z 673.559,A -85,B 0,C 180,E1 -9124.91,E2 -9124.91} C_VEL
LIN {X 0,Y 439.406,Z 663.916,A -85,B 0,C 180,E1 -9127.038,E2 -9127.038} C_VEL
LIN {X 0,Y 439.344,Z 663.528,A -85,B 0,C 180,E1 -9127.434,E2 -9127.434} C_VEL
LIN {X 0,Y 439.408,Z 663.561,A -85,B 0,C 180,E1 -9129.85,E2 -9129.85} C_VEL
LIN {X 0,Y 439.381,Z 663.567,A -85,B 0,C 180,E1 -9132.627,E2 -9132.627} C_VEL
LIN {X 0,Y 439.397,Z 663.566,A -85,B 0,C 180,E1 -9136.033,E2 -9136.033} C_VEL
LIN {X 0,Y 439.394,Z 663.544,A -85,B 0,C 180,E1 -9139.021,E2 -9139.021} C_VEL
LIN {X 0,Y 439.388,Z 663.568,A -85,B 0,C 180,E1 -9141.604,E2 -9141.604} C_VEL
LIN {X 0,Y 439.393,Z 663.545,A -85,B 0,C 180,E1 -9144.843,E2 -9144.843} C_VEL
LIN {X 0,Y 439.367,Z 663.565,A -85,B 0,C 180,E1 -9148.139,E2 -9148.139} C_VEL
LIN {X 0,Y 439.417,Z 663.52,A -85,B 0,C 180,E1 -9151.326,E2 -9151.326} C_VEL
LIN {X 0,Y 439.397,Z 663.562,A -85,B 0,C 180,E1 -9154.415,E2 -9154.415} C_VEL
LIN {X 0,Y 439.356,Z 663.556,A -85,B 0,C 180,E1 -9157.424,E2 -9157.424} C_VEL
LIN {X 0,Y 439.432,Z 663.557,A -85,B 0,C 180,E1 -9160.662,E2 -9160.662} C_VEL
LIN {X 0,Y 439.452,Z 663.555,A -85,B 0,C 180,E1 -9164.224,E2 -9164.224} C_VEL
LIN {X 0,Y 439.503,Z 663.542,A -85,B 0,C 180,E1 -9168.002,E2 -9168.002} C_VEL
LIN {X 0,Y 439.538,Z 663.53,A -85,B 0,C 180,E1 -9171.726,E2 -9171.726} C_VEL
LIN {X 0,Y 439.618,Z 663.532,A -85,B 0,C 180,E1 -9174.496,E2 -9174.496} C_VEL
LIN {X 0,Y 439.625,Z 663.527,A -85,B 0,C 180,E1 -9178.168,E2 -9178.168} C_VEL
LIN {X 0,Y 439.754,Z 663.516,A -85,B 0,C 180,E1 -9180,E2 -9180} C_VEL
LIN {X 0,Y 439.647,Z 663.517,A -85,B 0,C 180,E1 -9182.749,E2 -9182.749} C_VEL
LIN {X 0,Y 439.612,Z 663.53,A -85,B 0,C 180,E1 -9186.425,E2 -9186.425} C_VEL
LIN {X 0,Y 439.49,Z 663.546,A -85,B 0,C 180,E1 -9189.202,E2 -9189.202} C_VEL
LIN {X 0,Y 439.454,Z 663.541,A -85,B 0,C 180,E1 -9192.938,E2 -9192.938} C_VEL
LIN {X 0,Y 439.436,Z 663.553,A -85,B 0,C 180,E1 -9196.349,E2 -9196.349} C_VEL
LIN {X 0,Y 439.425,Z 663.557,A -85,B 0,C 180,E1 -9199.625,E2 -9199.625} C_VEL
LIN {X 0,Y 439.37,Z 663.56,A -85,B 0,C 180,E1 -9202.575,E2 -9202.575} C_VEL
LIN {X 0,Y 439.396,Z 663.56,A -85,B 0,C 180,E1 -9205.585,E2 -9205.585} C_VEL
LIN {X 0,Y 439.415,Z 663.526,A -85,B 0,C 180,E1 -9208.673,E2 -9208.673} C_VEL
LIN {X 0,Y 439.364,Z 663.564,A -85,B 0,C 180,E1 -9211.861,E2 -9211.861} C_VEL
LIN {X 0,Y 439.391,Z 663.539,A -85,B 0,C 180,E1 -9215.156,E2 -9215.156} C_VEL
LIN {X 0,Y 439.39,Z 663.56,A -85,B 0,C 180,E1 -9218.594,E2 -9218.594} C_VEL
LIN {X 0,Y 439.396,Z 663.567,A -85,B 0,C 180,E1 -9221.26,E2 -9221.26} C_VEL
LIN {X 0,Y 439.4,Z 663.565,A -85,B 0,C 180,E1 -9224.729,E2 -9224.729} C_VEL
LIN {X 0,Y 439.389,Z 663.566,A -85,B 0,C 180,E1 -9227.796,E2 -9227.796} C_VEL
LIN {X 0,Y 439.443,Z 663.557,A -85,B 0,C 180,E1 -9230.23,E2 -9230.23} C_VEL
LIN {X 0,Y 439.37,Z 663.57,A -85,B 0,C 180,E1 -9233.714,E2 -9233.714} C_VEL
LIN {X 0,Y 439.366,Z 663.568,A -85,B 0,C 180,E1 -9237.054,E2 -9237.054} C_VEL
LIN {X 0,Y 439.39,Z 663.567,A -85,B 0,C 180,E1 -9240.276,E2 -9240.276} C_VEL
LIN {X 0,Y 439.428,Z 663.563,A -85,B 0,C 180,E1 -9243.589,E2 -9243.589} C_VEL
LIN {X 0,Y 439.382,Z 663.567,A -85,B 0,C 180,E1 -9246.43,E2 -9246.43} C_VEL
LIN {X 0,Y 439.383,Z 663.565,A -85,B 0,C 180,E1 -9249.397,E2 -9249.397} C_VEL
LIN {X 0,Y 439.427,Z 663.562,A -85,B 0,C 180,E1 -9252.31,E2 -9252.31} C_VEL
LIN {X 0,Y 439.443,Z 663.56,A -85,B 0,C 180,E1 -9255.174,E2 -9255.174} C_VEL
LIN {X 0,Y 439.479,Z 663.555,A -85,B 0,C 180,E1 -9258.002,E2 -9258.002} C_VEL
LIN {X 0,Y 439.544,Z 663.546,A -85,B 0,C 180,E1 -9261.726,E2 -9261.726} C_VEL
LIN {X 0,Y 439.617,Z 663.538,A -85,B 0,C 180,E1 -9264.496,E2 -9264.496} C_VEL
LIN {X 0,Y 439.632,Z 663.534,A -85,B 0,C 180,E1 -9268.168,E2 -9268.168} C_VEL
LIN {X 0,Y 439.76,Z 663.52,A -85,B 0,C 180,E1 -9270,E2 -9270} C_VEL
LIN {X 0,Y 439.618,Z 663.537,A -85,B 0,C 180,E1 -9270.996,E2 -9270.996} C_VEL
LIN {X 0,Y 438.902,Z 663.626,A -85,B 0,C 180,E1 -9271.76,E2 -9271.76} C_VEL
LIN {X 0,Y 435.924,Z 663.999,A -85,B 0,C 180,E1 -9272.999,E2 -9272.999} C_VEL
LIN {X 0,Y 433.472,Z 664.304,A -85,B 0,C 180,E1 -9274,E2 -9274} C_VEL
LIN {X 0,Y 432.5,Z 664.424,A -85,B 0,C 180,E1 -9274.774,E2 -9274.774} C_VEL
LIN {X 0,Y 432.463,Z 664.427,A -85,B 0,C 180,E1 -9275.036,E2 -9275.036} C_VEL
LIN {X 0,Y 432.582,Z 664.415,A -85,B 0,C 180,E1 -9277.679,E2 -9277.679} C_VEL
LIN {X 0,Y 432.388,Z 664.438,A -85,B 0,C 180,E1 -9281.247,E2 -9281.247} C_VEL
LIN {X 0,Y 432.369,Z 664.44,A -85,B 0,C 180,E1 -9284.112,E2 -9284.112} C_VEL
LIN {X 0,Y 432.393,Z 664.436,A -85,B 0,C 180,E1 -9287.011,E2 -9287.011} C_VEL
LIN {X 0,Y 432.334,Z 664.447,A -85,B 0,C 180,E1 -9289.96,E2 -9289.96} C_VEL
LIN {X 0,Y 432.314,Z 664.447,A -85,B 0,C 180,E1 -9292.964,E2 -9292.964} C_VEL
LIN {X 0,Y 432.359,Z 664.442,A -85,B 0,C 180,E1 -9296.032,E2 -9296.032} C_VEL
LIN {X 0,Y 432.347,Z 664.442,A -85,B 0,C 180,E1 -9299.186,E2 -9299.186} C_VEL
LIN {X 0,Y 432.319,Z 664.449,A -85,B 0,C 180,E1 -9302.293,E2 -9302.293} C_VEL
LIN {X 0,Y 432.334,Z 664.447,A -85,B 0,C 180,E1 -9304.677,E2 -9304.677} C_VEL
LIN {X 0,Y 432.345,Z 664.445,A -85,B 0,C 180,E1 -9308.148,E2 -9308.148} C_VEL
LIN {X 0,Y 432.359,Z 664.44,A -85,B 0,C 180,E1 -9311.607,E2 -9311.607} C_VEL
LIN {X 0,Y 432.37,Z 664.438,A -85,B 0,C 180,E1 -9315.658,E2 -9315.658} C_VEL
LIN {X 0,Y 432.365,Z 664.44,A -85,B 0,C 180,E1 -9318.392,E2 -9318.392} C_VEL
LIN {X 0,Y 432.344,Z 664.434,A -85,B 0,C 180,E1 -9321.851,E2 -9321.851} C_VEL
LIN {X 0,Y 432.331,Z 664.425,A -85,B 0,C 180,E1 -9325.323,E2 -9325.323} C_VEL
LIN {X 0,Y 432.314,Z 664.443,A -85,B 0,C 180,E1 -9328.654,E2 -9328.654} C_VEL
LIN {X 0,Y 432.371,Z 664.402,A -85,B 0,C 180,E1 -9331.369,E2 -9331.369} C_VEL
LIN {X 0,Y 432.355,Z 664.435,A -85,B 0,C 180,E1 -9333.967,E2 -9333.967} C_VEL
LIN {X 0,Y 432.319,Z 664.44,A -85,B 0,C 180,E1 -9337.036,E2 -9337.036} C_VEL
LIN {X 0,Y 432.372,Z 664.44,A -85,B 0,C 180,E1 -9340.042,E2 -9340.042} C_VEL
LIN {X 0,Y 432.402,Z 664.427,A -85,B 0,C 180,E1 -9343.521,E2 -9343.521} C_VEL
LIN {X 0,Y 432.42,Z 664.416,A -85,B 0,C 180,E1 -9347.197,E2 -9347.197} C_VEL
LIN {X 0,Y 432.433,Z 664.425,A -85,B 0,C 180,E1 -9350.647,E2 -9350.647} C_VEL
LIN {X 0,Y 432.566,Z 664.407,A -85,B 0,C 180,E1 -9353.47,E2 -9353.47} C_VEL
LIN {X 0,Y 432.398,Z 664.431,A -85,B 0,C 180,E1 -9355.339,E2 -9355.339} C_VEL
LIN {X 0,Y 432.596,Z 664.398,A -85,B 0,C 180,E1 -9358.138,E2 -9358.138} C_VEL
LIN {X 0,Y 432.724,Z 664.393,A -85,B 0,C 180,E1 -9360,E2 -9360} C_VEL
LIN {X 0,Y 432.597,Z 664.4,A -85,B 0,C 180,E1 -9362.794,E2 -9362.794} C_VEL
LIN {X 0,Y 432.566,Z 664.414,A -85,B 0,C 180,E1 -9366.531,E2 -9366.531} C_VEL
LIN {X 0,Y 432.436,Z 664.429,A -85,B 0,C 180,E1 -9369.353,E2 -9369.353} C_VEL
LIN {X 0,Y 432.435,Z 664.42,A -85,B 0,C 180,E1 -9372.812,E2 -9372.812} C_VEL
LIN {X 0,Y 432.403,Z 664.43,A -85,B 0,C 180,E1 -9376.479,E2 -9376.479} C_VEL
LIN {X 0,Y 432.364,Z 664.439,A -85,B 0,C 180,E1 -9379.959,E2 -9379.959} C_VEL
LIN {X 0,Y 432.31,Z 664.435,A -85,B 0,C 180,E1 -9382.965,E2 -9382.965} C_VEL
LIN {X 0,Y 432.356,Z 664.432,A -85,B 0,C 180,E1 -9386.033,E2 -9386.033} C_VEL
LIN {X 0,Y 432.344,Z 664.401,A -85,B 0,C 180,E1 -9389.187,E2 -9389.187} C_VEL
LIN {X 0,Y 432.318,Z 664.447,A -85,B 0,C 180,E1 -9392.294,E2 -9392.294} C_VEL
LIN {X 0,Y 432.333,Z 664.427,A -85,B 0,C 180,E1 -9394.678,E2 -9394.678} C_VEL
LIN {X 0,Y 432.348,Z 664.442,A -85,B 0,C 180,E1 -9398.149,E2 -9398.149} C_VEL
LIN {X 0,Y 432.367,Z 664.42,A -85,B 0,C 180,E1 -9401.609,E2 -9401.609} C_VEL
LIN {X 0,Y 432.373,Z 664.432,A -85,B 0,C 180,E1 -9404.342,E2 -9404.342} C_VEL
LIN {X 0,Y 432.33,Z 664.439,A -85,B 0,C 180,E1 -9408.204,E2 -9408.204} C_VEL
LIN {X 0,Y 432.344,Z 664.431,A -85,B 0,C 180,E1 -9411.285,E2 -9411.285} C_VEL
LIN {X 0,Y 432.309,Z 664.519,A -85,B 0,C 180,E1 -9412.368,E2 -9412.368} C_VEL
LIN {X 0,Y 432.651,Z 665.889,A -85,B 0,C 180,E1 -9412.746,E2 -9412.746} C_VEL
LIN {X 0,Y 435.836,Z 677.514,A -85,B 0,C 180,E1 -9415.325,E2 -9415.325} C_VEL
LIN {X 0,Y 439.26,Z 691.744,A -85,B 0,C 180,E1 -9418.242,E2 -9418.242} C_VEL
LIN {X 0,Y 439.678,Z 693.208,A -85,B 0,C 180,E1 -9418.393,E2 -9418.393} C_VEL
LIN {X 0,Y 442.091,Z 701.525,A -85,B 0,C 180,E1 -9418.745,E2 -9418.745} C_VEL
LIN {X 0,Y 448.657,Z 728.798,A -85,B 0,C 180,E1 -9419.744,E2 -9419.744} C_VEL
LIN {X 0,Y 448.802,Z 733.059,A -85,B 0,C 180,E1 -9419.831,E2 -9419.831} C_VEL
LIN {X 0,Y 445.865,Z 894.4,A -85,B 0,C 180,E1 -9422.542,E2 -9422.542} C_VEL
LIN {X 0,Y 445.275,Z 906.703,A -85,B 0,C 180,E1 -9422.824,E2 -9422.824} C_VEL
LIN {X 0,Y 444.505,Z 920.043,A -85,B 0,C 180,E1 -9423.25,E2 -9423.25} C_VEL
LIN {X 0,Y 443.687,Z 933.167,A -85,B 0,C 180,E1 -9423.799,E2 -9423.799} C_VEL
LIN {X 0,Y 442.729,Z 944.554,A -85,B 0,C 180,E1 -9424.37,E2 -9424.37} C_VEL
LIN {X 0,Y 441.58,Z 958.157,A -85,B 0,C 180,E1 -9425.207,E2 -9425.207} C_VEL
LIN {X 0,Y 440.333,Z 970.539,A -85,B 0,C 180,E1 -9426.11,E2 -9426.11} C_VEL
LIN {X 0,Y 439.23,Z 981.541,A -85,B 0,C 180,E1 -9427.045,E2 -9427.045} C_VEL
LIN {X 0,Y 438.026,Z 992.345,A -85,B 0,C 180,E1 -9428.097,E2 -9428.097} C_VEL
LIN {X 0,Y 436.811,Z 1002.848,A -85,B 0,C 180,E1 -9429.271,E2 -9429.271} C_VEL
LIN {X 0,Y 435.856,Z 1012.124,A -85,B 0,C 180,E1 -9430.453,E2 -9430.453} C_VEL
LIN {X 0,Y 434.761,Z 1021.86,A -85,B 0,C 180,E1 -9431.87,E2 -9431.87} C_VEL
LIN {X 0,Y 433.904,Z 1030.387,A -85,B 0,C 180,E1 -9433.292,E2 -9433.292} C_VEL
LIN {X 0,Y 433.021,Z 1038.988,A -85,B 0,C 180,E1 -9434.949,E2 -9434.949} C_VEL
LIN {X 0,Y 432.489,Z 1045.419,A -85,B 0,C 180,E1 -9436.372,E2 -9436.372} C_VEL
LIN {X 0,Y 431.957,Z 1052.678,A -85,B 0,C 180,E1 -9438.266,E2 -9438.266} C_VEL
LIN {X 0,Y 431.617,Z 1057.324,A -85,B 0,C 180,E1 -9439.682,E2 -9439.682} C_VEL
LIN {X 0,Y 431.397,Z 1062.415,A -85,B 0,C 180,E1 -9441.569,E2 -9441.569} C_VEL
LIN {X 0,Y 431.293,Z 1066.406,A -85,B 0,C 180,E1 -9443.45,E2 -9443.45} C_VEL
LIN {X 0,Y 431.21,Z 1069.352,A -85,B 0,C 180,E1 -9445.326,E2 -9445.326} C_VEL
LIN {X 0,Y 431.143,Z 1070.533,A -85,B 0,C 180,E1 -9446.262,E2 -9446.262} C_VEL
LIN {X 0,Y 431.192,Z 1071.996,A -85,B 0,C 180,E1 -9448.132,E2 -9448.132} C_VEL
LIN {X 0,Y 431.163,Z 1072.48,A -85,B 0,C 180,E1 -9450,E2 -9450} C_VEL
LIN {X 0,Y 431.192,Z 1071.996,A -85,B 0,C 180,E1 -9451.868,E2 -9451.868} C_VEL
LIN {X 0,Y 431.143,Z 1070.533,A -85,B 0,C 180,E1 -9453.738,E2 -9453.738} C_VEL
LIN {X 0,Y 431.224,Z 1068.075,A -85,B 0,C 180,E1 -9455.612,E2 -9455.612} C_VEL
LIN {X 0,Y 431.375,Z 1063.502,A -85,B 0,C 180,E1 -9457.96,E2 -9457.96} C_VEL
LIN {X 0,Y 431.489,Z 1060.018,A -85,B 0,C 180,E1 -9459.374,E2 -9459.374} C_VEL
LIN {X 0,Y 431.845,Z 1054.298,A -85,B 0,C 180,E1 -9461.261,E2 -9461.261} C_VEL
LIN {X 0,Y 432.196,Z 1049.3,A -85,B 0,C 180,E1 -9462.666,E2 -9462.666} C_VEL
LIN {X 0,Y 432.845,Z 1041.211,A -85,B 0,C 180,E1 -9464.576,E2 -9464.576} C_VEL
LIN {X 0,Y 433.589,Z 1034.229,A -85,B 0,C 180,E1 -9465.994,E2 -9465.994} C_VEL
LIN {X 0,Y 434.342,Z 1026.045,A -85,B 0,C 180,E1 -9467.453,E2 -9467.453} C_VEL
LIN {X 0,Y 435.276,Z 1017.141,A -85,B 0,C 180,E1 -9468.839,E2 -9468.839} C_VEL
LIN {X 0,Y 436.195,Z 1008.569,A -85,B 0,C 180,E1 -9470.021,E2 -9470.021} C_VEL
LIN {X 0,Y 437.424,Z 998.174,A -85,B 0,C 180,E1 -9471.272,E2 -9471.272} C_VEL
LIN {X 0,Y 438.674,Z 986.53,A -85,B 0,C 180,E1 -9472.488,E2 -9472.488} C_VEL
LIN {X 0,Y 439.844,Z 974.853,A -85,B 0,C 180,E1 -9473.544,E2 -9473.544} C_VEL
LIN {X 0,Y 441.13,Z 962.826,A -85,B 0,C 180,E1 -9474.47,E2 -9474.47} C_VEL
LIN {X 0,Y 442.302,Z 950.066,A -85,B 0,C 180,E1 -9475.306,E2 -9475.306} C_VEL
LIN {X 0,Y 443.314,Z 937.954,A -85,B 0,C 180,E1 -9475.972,E2 -9475.972} C_VEL
LIN {X 0,Y 444.257,Z 925.27,A -85,B 0,C 180,E1 -9476.545,E2 -9476.545} C_VEL
LIN {X 0,Y 444.978,Z 911.599,A -85,B 0,C 180,E1 -9477.037,E2 -9477.037} C_VEL
LIN {X 0,Y 445.691,Z 897.945,A -85,B 0,C 180,E1 -9477.389,E2 -9477.389} C_VEL
LIN {X 0,Y 446.282,Z 873.197,A -85,B 0,C 180,E1 -9477.832,E2 -9477.832} C_VEL
LIN {X 0,Y 448.853,Z 730.107,A -85,B 0,C 180,E1 -9480.218,E2 -9480.218} C_VEL
LIN {X 0,Y 444.097,Z 709.46,A -85,B 0,C 180,E1 -9480.953,E2 -9480.953} C_VEL
LIN {X 0,Y 440.139,Z 694.424,A -85,B 0,C 180,E1 -9481.541,E2 -9481.541} C_VEL
LIN {X 0,Y 439.323,Z 692.136,A -85,B 0,C 180,E1 -9481.696,E2 -9481.696} C_VEL
LIN {X 0,Y 435.855,Z 677.486,A -85,B 0,C 180,E1 -9484.679,E2 -9484.679} C_VEL
LIN {X 0,Y 432.389,Z 664.875,A -85,B 0,C 180,E1 -9487.495,E2 -9487.495} C_VEL
LIN {X 0,Y 432.308,Z 664.425,A -85,B 0,C 180,E1 -9487.762,E2 -9487.762} C_VEL
LIN {X 0,Y 432.323,Z 664.435,A -85,B 0,C 180,E1 -9490.559,E2 -9490.559} C_VEL
LIN {X 0,Y 432.318,Z 664.445,A -85,B 0,C 180,E1 -9493.059,E2 -9493.059} C_VEL
LIN {X 0,Y 432.373,Z 664.432,A -85,B 0,C 180,E1 -9495.658,E2 -9495.658} C_VEL
LIN {X 0,Y 432.367,Z 664.42,A -85,B 0,C 180,E1 -9498.391,E2 -9498.391} C_VEL
LIN {X 0,Y 432.348,Z 664.442,A -85,B 0,C 180,E1 -9501.851,E2 -9501.851} C_VEL
LIN {X 0,Y 432.333,Z 664.427,A -85,B 0,C 180,E1 -9505.322,E2 -9505.322} C_VEL
LIN {X 0,Y 432.316,Z 664.437,A -85,B 0,C 180,E1 -9508.653,E2 -9508.653} C_VEL
LIN {X 0,Y 432.373,Z 664.396,A -85,B 0,C 180,E1 -9511.368,E2 -9511.368} C_VEL
LIN {X 0,Y 432.356,Z 664.432,A -85,B 0,C 180,E1 -9513.967,E2 -9513.967} C_VEL
LIN {X 0,Y 432.31,Z 664.435,A -85,B 0,C 180,E1 -9517.035,E2 -9517.035} C_VEL
LIN {X 0,Y 432.382,Z 664.438,A -85,B 0,C 180,E1 -9520.513,E2 -9520.513} C_VEL
LIN {X 0,Y 432.421,Z 664.429,A -85,B 0,C 180,E1 -9523.961,E2 -9523.961} C_VEL
LIN {X 0,Y 432.475,Z 664.417,A -85,B 0,C 180,E1 -9527.804,E2 -9527.804} C_VEL
LIN {X 0,Y 432.482,Z 664.41,A -85,B 0,C 180,E1 -9531.59,E2 -9531.59} C_VEL
LIN {X 0,Y 432.594,Z 664.407,A -85,B 0,C 180,E1 -9534.406,E2 -9534.406} C_VEL
LIN {X 0,Y 432.596,Z 664.402,A -85,B 0,C 180,E1 -9538.138,E2 -9538.138} C_VEL
LIN {X 0,Y 432.724,Z 664.392,A -85,B 0,C 180,E1 -9540,E2 -9540} C_VEL
LIN {X 0,Y 432.597,Z 664.395,A -85,B 0,C 180,E1 -9542.793,E2 -9542.793} C_VEL
LIN {X 0,Y 432.566,Z 664.408,A -85,B 0,C 180,E1 -9546.53,E2 -9546.53} C_VEL
LIN {X 0,Y 432.433,Z 664.426,A -85,B 0,C 180,E1 -9549.353,E2 -9549.353} C_VEL
LIN {X 0,Y 432.42,Z 664.417,A -85,B 0,C 180,E1 -9552.803,E2 -9552.803} C_VEL
LIN {X 0,Y 432.402,Z 664.428,A -85,B 0,C 180,E1 -9556.479,E2 -9556.479} C_VEL
LIN {X 0,Y 432.372,Z 664.44,A -85,B 0,C 180,E1 -9559.958,E2 -9559.958} C_VEL
LIN {X 0,Y 432.319,Z 664.44,A -85,B 0,C 180,E1 -9562.964,E2 -9562.964} C_VEL
LIN {X 0,Y 432.355,Z 664.435,A -85,B 0,C 180,E1 -9566.033,E2 -9566.033} C_VEL
LIN {X 0,Y 432.342,Z 664.407,A -85,B 0,C 180,E1 -9569.187,E2 -9569.187} C_VEL
LIN {X 0,Y 432.316,Z 664.445,A -85,B 0,C 180,E1 -9572.294,E2 -9572.294} C_VEL
LIN {X 0,Y 432.331,Z 664.425,A -85,B 0,C 180,E1 -9574.677,E2 -9574.677} C_VEL
LIN {X 0,Y 432.344,Z 664.434,A -85,B 0,C 180,E1 -9578.149,E2 -9578.149} C_VEL
LIN {X 0,Y 432.365,Z 664.44,A -85,B 0,C 180,E1 -9581.608,E2 -9581.608} C_VEL
LIN {X 0,Y 432.37,Z 664.438,A -85,B 0,C 180,E1 -9584.342,E2 -9584.342} C_VEL
LIN {X 0,Y 432.359,Z 664.44,A -85,B 0,C 180,E1 -9588.393,E2 -9588.393} C_VEL
LIN {X 0,Y 432.345,Z 664.445,A -85,B 0,C 180,E1 -9591.852,E2 -9591.852} C_VEL
LIN {X 0,Y 432.334,Z 664.447,A -85,B 0,C 180,E1 -9595.323,E2 -9595.323} C_VEL
LIN {X 0,Y 432.318,Z 664.445,A -85,B 0,C 180,E1 -9598.655,E2 -9598.655} C_VEL
LIN {X 0,Y 432.375,Z 664.439,A -85,B 0,C 180,E1 -9601.369,E2 -9601.369} C_VEL
LIN {X 0,Y 432.359,Z 664.442,A -85,B 0,C 180,E1 -9603.968,E2 -9603.968} C_VEL
LIN {X 0,Y 432.314,Z 664.447,A -85,B 0,C 180,E1 -9607.036,E2 -9607.036} C_VEL
LIN {X 0,Y 432.382,Z 664.438,A -85,B 0,C 180,E1 -9610.515,E2 -9610.515} C_VEL
LIN {X 0,Y 432.426,Z 664.434,A -85,B 0,C 180,E1 -9613.961,E2 -9613.961} C_VEL
LIN {X 0,Y 432.455,Z 664.429,A -85,B 0,C 180,E1 -9617.804,E2 -9617.804} C_VEL
LIN {X 0,Y 432.488,Z 664.425,A -85,B 0,C 180,E1 -9621.59,E2 -9621.59} C_VEL
LIN {X 0,Y 432.594,Z 664.412,A -85,B 0,C 180,E1 -9624.406,E2 -9624.406} C_VEL
LIN {X 0,Y 432.602,Z 664.41,A -85,B 0,C 180,E1 -9628.138,E2 -9628.138} C_VEL
LIN {X 0,Y 432.73,Z 664.396,A -85,B 0,C 180,E1 -9630,E2 -9630} C_VEL
LIN {X 0,Y 432.602,Z 664.414,A -85,B 0,C 180,E1 -9632.793,E2 -9632.793} C_VEL
LIN {X 0,Y 432.463,Z 664.427,A -85,B 0,C 180,E1 -9635.036,E2 -9635.036} C_VEL
LIN {X 0,Y 431.903,Z 664.498,A -85,B 0,C 180,E1 -9635.815,E2 -9635.815} C_VEL
LIN {X 0,Y 429.056,Z 664.853,A -85,B 0,C 180,E1 -9637.08,E2 -9637.08} C_VEL
LIN {X 0,Y 426.571,Z 665.163,A -85,B 0,C 180,E1 -9638.101,E2 -9638.101} C_VEL
LIN {X 0,Y 425.49,Z 665.297,A -85,B 0,C 180,E1 -9638.891,E2 -9638.891} C_VEL
LIN {X 0,Y 425.399,Z 665.307,A -85,B 0,C 180,E1 -9639.158,E2 -9639.158} C_VEL
LIN {X 0,Y 425.389,Z 665.309,A -85,B 0,C 180,E1 -9642.903,E2 -9642.903} C_VEL
LIN {X 0,Y 425.357,Z 665.312,A -85,B 0,C 180,E1 -9646.605,E2 -9646.605} C_VEL
LIN {X 0,Y 425.324,Z 665.318,A -85,B 0,C 180,E1 -9649.635,E2 -9649.635} C_VEL
LIN {X 0,Y 425.302,Z 665.32,A -85,B 0,C 180,E1 -9653.365,E2 -9653.365} C_VEL
LIN {X 0,Y 425.343,Z 665.315,A -85,B 0,C 180,E1 -9656.844,E2 -9656.844} C_VEL
LIN {X 0,Y 425.312,Z 665.321,A -85,B 0,C 180,E1 -9659.717,E2 -9659.717} C_VEL
LIN {X 0,Y 425.276,Z 665.324,A -85,B 0,C 180,E1 -9663.048,E2 -9663.048} C_VEL
LIN {X 0,Y 425.278,Z 665.323,A -85,B 0,C 180,E1 -9665.929,E2 -9665.929} C_VEL
LIN {X 0,Y 425.305,Z 665.321,A -85,B 0,C 180,E1 -9669.045,E2 -9669.045} C_VEL
LIN {X 0,Y 425.307,Z 665.319,A -85,B 0,C 180,E1 -9671.962,E2 -9671.962} C_VEL
LIN {X 0,Y 425.305,Z 665.321,A -85,B 0,C 180,E1 -9675.279,E2 -9675.279} C_VEL
LIN {X 0,Y 425.302,Z 665.322,A -85,B 0,C 180,E1 -9678.625,E2 -9678.625} C_VEL
LIN {X 0,Y 425.315,Z 665.317,A -85,B 0,C 180,E1 -9681.104,E2 -9681.104} C_VEL
LIN {X 0,Y 425.291,Z 665.292,A -85,B 0,C 180,E1 -9684.664,E2 -9684.664} C_VEL
LIN {X 0,Y 425.256,Z 665.322,A -85,B 0,C 180,E1 -9688.073,E2 -9688.073} C_VEL
LIN {X 0,Y 425.328,Z 665.277,A -85,B 0,C 180,E1 -9691.368,E2 -9691.368} C_VEL
LIN {X 0,Y 425.286,Z 665.318,A -85,B 0,C 180,E1 -9694.555,E2 -9694.555} C_VEL
LIN {X 0,Y 425.313,Z 665.31,A -85,B 0,C 180,E1 -9697.719,E2 -9697.719} C_VEL
LIN {X 0,Y 425.355,Z 665.309,A -85,B 0,C 180,E1 -9700.704,E2 -9700.704} C_VEL
LIN {X 0,Y 425.378,Z 665.304,A -85,B 0,C 180,E1 -9703.688,E2 -9703.688} C_VEL
LIN {X 0,Y 425.402,Z 665.291,A -85,B 0,C 180,E1 -9707.598,E2 -9707.598} C_VEL
LIN {X 0,Y 425.432,Z 665.294,A -85,B 0,C 180,E1 -9711.45,E2 -9711.45} C_VEL
LIN {X 0,Y 425.569,Z 665.285,A -85,B 0,C 180,E1 -9714.314,E2 -9714.314} C_VEL
LIN {X 0,Y 425.566,Z 665.273,A -85,B 0,C 180,E1 -9718.108,E2 -9718.108} C_VEL
LIN {X 0,Y 425.694,Z 665.269,A -85,B 0,C 180,E1 -9720,E2 -9720} C_VEL
LIN {X 0,Y 425.549,Z 665.278,A -85,B 0,C 180,E1 -9722.84,E2 -9722.84} C_VEL
LIN {X 0,Y 425.569,Z 665.282,A -85,B 0,C 180,E1 -9725.687,E2 -9725.687} C_VEL
LIN {X 0,Y 425.433,Z 665.287,A -85,B 0,C 180,E1 -9728.55,E2 -9728.55} C_VEL
LIN {X 0,Y 425.423,Z 665.295,A -85,B 0,C 180,E1 -9732.402,E2 -9732.402} C_VEL
LIN {X 0,Y 425.379,Z 665.305,A -85,B 0,C 180,E1 -9736.312,E2 -9736.312} C_VEL
LIN {X 0,Y 425.352,Z 665.316,A -85,B 0,C 180,E1 -9739.648,E2 -9739.648} C_VEL
LIN {X 0,Y 425.298,Z 665.312,A -85,B 0,C 180,E1 -9743.366,E2 -9743.366} C_VEL
LIN {X 0,Y 425.341,Z 665.301,A -85,B 0,C 180,E1 -9746.845,E2 -9746.845} C_VEL
LIN {X 0,Y 425.31,Z 665.281,A -85,B 0,C 180,E1 -9749.718,E2 -9749.718} C_VEL
LIN {X 0,Y 425.275,Z 665.321,A -85,B 0,C 180,E1 -9753.049,E2 -9753.049} C_VEL
LIN {X 0,Y 425.277,Z 665.298,A -85,B 0,C 180,E1 -9755.93,E2 -9755.93} C_VEL
LIN {X 0,Y 425.309,Z 665.317,A -85,B 0,C 180,E1 -9759.047,E2 -9759.047} C_VEL
LIN {X 0,Y 425.326,Z 665.311,A -85,B 0,C 180,E1 -9762.647,E2 -9762.647} C_VEL
LIN {X 0,Y 425.294,Z 665.303,A -85,B 0,C 180,E1 -9765.282,E2 -9765.282} C_VEL
LIN {X 0,Y 425.271,Z 665.313,A -85,B 0,C 180,E1 -9768.622,E2 -9768.622} C_VEL
LIN {X 0,Y 425.324,Z 665.37,A -85,B 0,C 180,E1 -9771.862,E2 -9771.862} C_VEL
LIN {X 0,Y 425.781,Z 667.411,A -85,B 0,C 180,E1 -9772.4,E2 -9772.4} C_VEL
LIN {X 0,Y 429.217,Z 680.023,A -85,B 0,C 180,E1 -9775.25,E2 -9775.25} C_VEL
LIN {X 0,Y 432.14,Z 692.16,A -85,B 0,C 180,E1 -9777.746,E2 -9777.746} C_VEL
LIN {X 0,Y 434.753,Z 698.29,A -85,B 0,C 180,E1 -9778.099,E2 -9778.099} C_VEL
LIN {X 0,Y 441.504,Z 725.652,A -85,B 0,C 180,E1 -9779.147,E2 -9779.147} C_VEL
LIN {X 0,Y 442.7,Z 731.614,A -85,B 0,C 180,E1 -9779.348,E2 -9779.348} C_VEL
LIN {X 0,Y 439.558,Z 894.544,A -85,B 0,C 180,E1 -9782.122,E2 -9782.122} C_VEL
LIN {X 0,Y 438.916,Z 907.477,A -85,B 0,C 180,E1 -9782.429,E2 -9782.429} C_VEL
LIN {X 0,Y 438.168,Z 919.837,A -85,B 0,C 180,E1 -9782.831,E2 -9782.831} C_VEL
LIN {X 0,Y 437.286,Z 932.96,A -85,B 0,C 180,E1 -9783.385,E2 -9783.385} C_VEL
LIN {X 0,Y 436.3,Z 944.348,A -85,B 0,C 180,E1 -9783.964,E2 -9783.964} C_VEL
LIN {X 0,Y 435.143,Z 957.27,A -85,B 0,C 180,E1 -9784.764,E2 -9784.764} C_VEL
LIN {X 0,Y 433.953,Z 968.893,A -85,B 0,C 180,E1 -9785.609,E2 -9785.609} C_VEL
LIN {X 0,Y 432.644,Z 981.334,A -85,B 0,C 180,E1 -9786.675,E2 -9786.675} C_VEL
LIN {X 0,Y 431.365,Z 992.137,A -85,B 0,C 180,E1 -9787.741,E2 -9787.741} C_VEL
LIN {X 0,Y 430.108,Z 1002.64,A -85,B 0,C 180,E1 -9788.932,E2 -9788.932} C_VEL
LIN {X 0,Y 429.061,Z 1011.915,A -85,B 0,C 180,E1 -9790.131,E2 -9790.131} C_VEL
LIN {X 0,Y 427.903,Z 1021.651,A -85,B 0,C 180,E1 -9791.569,E2 -9791.569} C_VEL
LIN {X 0,Y 426.96,Z 1030.177,A -85,B 0,C 180,E1 -9793.012,E2 -9793.012} C_VEL
LIN {X 0,Y 426.051,Z 1038.779,A -85,B 0,C 180,E1 -9794.697,E2 -9794.697} C_VEL
LIN {X 0,Y 425.501,Z 1045.211,A -85,B 0,C 180,E1 -9796.144,E2 -9796.144} C_VEL
LIN {X 0,Y 424.941,Z 1052.47,A -85,B 0,C 180,E1 -9798.069,E2 -9798.069} C_VEL
LIN {X 0,Y 424.58,Z 1057.117,A -85,B 0,C 180,E1 -9799.509,E2 -9799.509} C_VEL
LIN {X 0,Y 424.335,Z 1062.209,A -85,B 0,C 180,E1 -9801.428,E2 -9801.428} C_VEL
LIN {X 0,Y 424.214,Z 1066.2,A -85,B 0,C 180,E1 -9803.341,E2 -9803.341} C_VEL
LIN {X 0,Y 424.136,Z 1069.147,A -85,B 0,C 180,E1 -9805.248,E2 -9805.248} C_VEL
LIN {X 0,Y 424.055,Z 1070.327,A -85,B 0,C 180,E1 -9806.199,E2 -9806.199} C_VEL
LIN {X 0,Y 424.118,Z 1071.792,A -85,B 0,C 180,E1 -9808.101,E2 -9808.101} C_VEL
LIN {X 0,Y 424.08,Z 1072.275,A -85,B 0,C 180,E1 -9810,E2 -9810} C_VEL
LIN {X 0,Y 424.118,Z 1071.792,A -85,B 0,C 180,E1 -9811.899,E2 -9811.899} C_VEL
LIN {X 0,Y 424.055,Z 1070.327,A -85,B 0,C 180,E1 -9813.801,E2 -9813.801} C_VEL
LIN {X 0,Y 424.143,Z 1067.869,A -85,B 0,C 180,E1 -9815.706,E2 -9815.706} C_VEL
LIN {X 0,Y 424.282,Z 1063.295,A -85,B 0,C 180,E1 -9818.094,E2 -9818.094} C_VEL
LIN {X 0,Y 424.401,Z 1059.81,A -85,B 0,C 180,E1 -9819.532,E2 -9819.532} C_VEL
LIN {X 0,Y 424.787,Z 1054.09,A -85,B 0,C 180,E1 -9821.451,E2 -9821.451} C_VEL
LIN {X 0,Y 425.21,Z 1048.72,A -85,B 0,C 180,E1 -9822.972,E2 -9822.972} C_VEL
LIN {X 0,Y 425.849,Z 1041.001,A -85,B 0,C 180,E1 -9824.821,E2 -9824.821} C_VEL
LIN {X 0,Y 426.667,Z 1034.021,A -85,B 0,C 180,E1 -9826.261,E2 -9826.261} C_VEL
LIN {X 0,Y 427.424,Z 1026.218,A -85,B 0,C 180,E1 -9827.68,E2 -9827.68} C_VEL
LIN {X 0,Y 428.441,Z 1016.932,A -85,B 0,C 180,E1 -9829.151,E2 -9829.151} C_VEL
LIN {X 0,Y 429.451,Z 1008.361,A -85,B 0,C 180,E1 -9830.35,E2 -9830.35} C_VEL
LIN {X 0,Y 430.87,Z 996.583,A -85,B 0,C 180,E1 -9831.771,E2 -9831.771} C_VEL
LIN {X 0,Y 432.064,Z 986.323,A -85,B 0,C 180,E1 -9832.851,E2 -9832.851} C_VEL
LIN {X 0,Y 433.292,Z 974.646,A -85,B 0,C 180,E1 -9833.922,E2 -9833.922} C_VEL
LIN {X 0,Y 434.621,Z 962.618,A -85,B 0,C 180,E1 -9834.861,E2 -9834.861} C_VEL
LIN {X 0,Y 435.826,Z 950.007,A -85,B 0,C 180,E1 -9835.7,E2 -9835.7} C_VEL
LIN {X 0,Y 436.911,Z 937.747,A -85,B 0,C 180,E1 -9836.382,E2 -9836.382} C_VEL
LIN {X 0,Y 437.926,Z 924.317,A -85,B 0,C 180,E1 -9836.991,E2 -9836.991} C_VEL
LIN {X 0,Y 438.658,Z 911.393,A -85,B 0,C 180,E1 -9837.459,E2 -9837.459} C_VEL
LIN {X 0,Y 439.394,Z 898.04,A -85,B 0,C 180,E1 -9837.809,E2 -9837.809} C_VEL
LIN {X 0,Y 440.005,Z 873.034,A -85,B 0,C 180,E1 -9838.264,E2 -9838.264} C_VEL
LIN {X 0,Y 442.672,Z 730.668,A -85,B 0,C 180,E1 -9840.671,E2 -9840.671} C_VEL
LIN {X 0,Y 435.92,Z 702.6,A -85,B 0,C 180,E1 -9841.725,E2 -9841.725} C_VEL
LIN {X 0,Y 433.938,Z 696.105,A -85,B 0,C 180,E1 -9842.009,E2 -9842.009} C_VEL
LIN {X 0,Y 432.059,Z 692.006,A -85,B 0,C 180,E1 -9842.274,E2 -9842.274} C_VEL
LIN {X 0,Y 428.957,Z 678.871,A -85,B 0,C 180,E1 -9844.996,E2 -9844.996} C_VEL
LIN {X 0,Y 425.319,Z 665.525,A -85,B 0,C 180,E1 -9848.064,E2 -9848.064} C_VEL
LIN {X 0,Y 425.296,Z 665.318,A -85,B 0,C 180,E1 -9849.043,E2 -9849.043} C_VEL
LIN {X 0,Y 425.273,Z 665.325,A -85,B 0,C 180,E1 -9852.652,E2 -9852.652} C_VEL
LIN {X 0,Y 425.329,Z 665.317,A -85,B 0,C 180,E1 -9856.053,E2 -9856.053} C_VEL
LIN {X 0,Y 425.304,Z 665.298,A -85,B 0,C 180,E1 -9858.625,E2 -9858.625} C_VEL
LIN {X 0,Y 425.32,Z 665.316,A -85,B 0,C 180,E1 -9861.104,E2 -9861.104} C_VEL
LIN {X 0,Y 425.293,Z 665.297,A -85,B 0,C 180,E1 -9864.663,E2 -9864.663} C_VEL
LIN {X 0,Y 425.259,Z 665.323,A -85,B 0,C 180,E1 -9868.073,E2 -9868.073} C_VEL
LIN {X 0,Y 425.33,Z 665.272,A -85,B 0,C 180,E1 -9871.368,E2 -9871.368} C_VEL
LIN {X 0,Y 425.288,Z 665.322,A -85,B 0,C 180,E1 -9874.554,E2 -9874.554} C_VEL
LIN {X 0,Y 425.279,Z 665.309,A -85,B 0,C 180,E1 -9877.661,E2 -9877.661} C_VEL
LIN {X 0,Y 425.355,Z 665.31,A -85,B 0,C 180,E1 -9880.704,E2 -9880.704} C_VEL
LIN {X 0,Y 425.379,Z 665.306,A -85,B 0,C 180,E1 -9883.688,E2 -9883.688} C_VEL
LIN {X 0,Y 425.423,Z 665.296,A -85,B 0,C 180,E1 -9887.598,E2 -9887.598} C_VEL
LIN {X 0,Y 425.433,Z 665.288,A -85,B 0,C 180,E1 -9891.45,E2 -9891.45} C_VEL
LIN {X 0,Y 425.569,Z 665.282,A -85,B 0,C 180,E1 -9894.313,E2 -9894.313} C_VEL
LIN {X 0,Y 425.565,Z 665.278,A -85,B 0,C 180,E1 -9898.107,E2 -9898.107} C_VEL
LIN {X 0,Y 425.694,Z 665.268,A -85,B 0,C 180,E1 -9900,E2 -9900} C_VEL
LIN {X 0,Y 425.549,Z 665.273,A -85,B 0,C 180,E1 -9902.84,E2 -9902.84} C_VEL
LIN {X 0,Y 425.569,Z 665.286,A -85,B 0,C 180,E1 -9905.686,E2 -9905.686} C_VEL
LIN {X 0,Y 425.432,Z 665.295,A -85,B 0,C 180,E1 -9908.55,E2 -9908.55} C_VEL
LIN {X 0,Y 425.402,Z 665.292,A -85,B 0,C 180,E1 -9912.402,E2 -9912.402} C_VEL
LIN {X 0,Y 425.378,Z 665.304,A -85,B 0,C 180,E1 -9916.312,E2 -9916.312} C_VEL
LIN {X 0,Y 425.352,Z 665.311,A -85,B 0,C 180,E1 -9919.649,E2 -9919.649} C_VEL
LIN {X 0,Y 425.294,Z 665.312,A -85,B 0,C 180,E1 -9922.338,E2 -9922.338} C_VEL
LIN {X 0,Y 425.286,Z 665.318,A -85,B 0,C 180,E1 -9925.445,E2 -9925.445} C_VEL
LIN {X 0,Y 425.328,Z 665.277,A -85,B 0,C 180,E1 -9928.632,E2 -9928.632} C_VEL
LIN {X 0,Y 425.256,Z 665.322,A -85,B 0,C 180,E1 -9931.927,E2 -9931.927} C_VEL
LIN {X 0,Y 425.291,Z 665.292,A -85,B 0,C 180,E1 -9935.336,E2 -9935.336} C_VEL
LIN {X 0,Y 425.305,Z 665.321,A -85,B 0,C 180,E1 -9939.046,E2 -9939.046} C_VEL
LIN {X 0,Y 425.323,Z 665.319,A -85,B 0,C 180,E1 -9942.646,E2 -9942.646} C_VEL
LIN {X 0,Y 425.286,Z 665.325,A -85,B 0,C 180,E1 -9945.282,E2 -9945.282} C_VEL
LIN {X 0,Y 425.296,Z 665.32,A -85,B 0,C 180,E1 -9948.625,E2 -9948.625} C_VEL
LIN {X 0,Y 425.316,Z 665.321,A -85,B 0,C 180,E1 -9951.104,E2 -9951.104} C_VEL
LIN {X 0,Y 425.294,Z 665.32,A -85,B 0,C 180,E1 -9954.665,E2 -9954.665} C_VEL
LIN {X 0,Y 425.26,Z 665.326,A -85,B 0,C 180,E1 -9958.074,E2 -9958.074} C_VEL
LIN {X 0,Y 425.332,Z 665.316,A -85,B 0,C 180,E1 -9961.369,E2 -9961.369} C_VEL
LIN {X 0,Y 425.29,Z 665.323,A -85,B 0,C 180,E1 -9964.555,E2 -9964.555} C_VEL
LIN {X 0,Y 425.283,Z 665.324,A -85,B 0,C 180,E1 -9967.662,E2 -9967.662} C_VEL
LIN {X 0,Y 425.357,Z 665.313,A -85,B 0,C 180,E1 -9970.704,E2 -9970.704} C_VEL
LIN {X 0,Y 425.384,Z 665.309,A -85,B 0,C 180,E1 -9973.689,E2 -9973.689} C_VEL
LIN {X 0,Y 425.408,Z 665.306,A -85,B 0,C 180,E1 -9977.598,E2 -9977.598} C_VEL
LIN {X 0,Y 425.439,Z 665.302,A -85,B 0,C 180,E1 -9981.45,E2 -9981.45} C_VEL
LIN {X 0,Y 425.55,Z 665.289,A -85,B 0,C 180,E1 -9984.313,E2 -9984.313} C_VEL
LIN {X 0,Y 425.572,Z 665.286,A -85,B 0,C 180,E1 -9988.107,E2 -9988.107} C_VEL
LIN {X 0,Y 425.7,Z 665.272,A -85,B 0,C 180,E1 -9990,E2 -9990} C_VEL
LIN {X 0,Y 425.553,Z 665.291,A -85,B 0,C 180,E1 -9992.84,E2 -9992.84} C_VEL
LIN {X 0,Y 425.527,Z 665.294,A -85,B 0,C 180,E1 -9996.639,E2 -9996.639} C_VEL
LIN {X 0,Y 425.399,Z 665.307,A -85,B 0,C 180,E1 -9999.158,E2 -9999.158} C_VEL
LIN {X 0,Y 424.727,Z 665.393,A -85,B 0,C 180,E1 -9999.948,E2 -9999.948} C_VEL
LIN {X 0,Y 421.878,Z 665.748,A -85,B 0,C 180,E1 -10001.232,E2 -10001.232} C_VEL
LIN {X 0,Y 419.462,Z 666.048,A -85,B 0,C 180,E1 -10002.268,E2 -10002.268} C_VEL
LIN {X 0,Y 418.411,Z 666.179,A -85,B 0,C 180,E1 -10003.069,E2 -10003.069} C_VEL
LIN {X 0,Y 418.318,Z 666.19,A -85,B 0,C 180,E1 -10003.34,E2 -10003.34} C_VEL
LIN {X 0,Y 418.308,Z 666.19,A -85,B 0,C 180,E1 -10006.735,E2 -10006.735} C_VEL
LIN {X 0,Y 418.266,Z 666.198,A -85,B 0,C 180,E1 -10009.79,E2 -10009.79} C_VEL
LIN {X 0,Y 418.233,Z 666.202,A -85,B 0,C 180,E1 -10012.736,E2 -10012.736} C_VEL
LIN {X 0,Y 418.266,Z 666.198,A -85,B 0,C 180,E1 -10015.904,E2 -10015.904} C_VEL
LIN {X 0,Y 418.269,Z 666.196,A -85,B 0,C 180,E1 -10019.161,E2 -10019.161} C_VEL
LIN {X 0,Y 418.251,Z 666.198,A -85,B 0,C 180,E1 -10022.844,E2 -10022.844} C_VEL
LIN {X 0,Y 418.242,Z 666.201,A -85,B 0,C 180,E1 -10026.238,E2 -10026.238} C_VEL
LIN {X 0,Y 418.258,Z 666.196,A -85,B 0,C 180,E1 -10029.68,E2 -10029.68} C_VEL
LIN {X 0,Y 418.237,Z 666.202,A -85,B 0,C 180,E1 -10032.323,E2 -10032.323} C_VEL
LIN {X 0,Y 418.25,Z 666.201,A -85,B 0,C 180,E1 -10035.111,E2 -10035.111} C_VEL
LIN {X 0,Y 418.284,Z 666.193,A -85,B 0,C 180,E1 -10037.773,E2 -10037.773} C_VEL
LIN {X 0,Y 418.258,Z 666.19,A -85,B 0,C 180,E1 -10041.559,E2 -10041.559} C_VEL
LIN {X 0,Y 418.25,Z 666.174,A -85,B 0,C 180,E1 -10045.159,E2 -10045.159} C_VEL
LIN {X 0,Y 418.236,Z 666.202,A -85,B 0,C 180,E1 -10047.472,E2 -10047.472} C_VEL
LIN {X 0,Y 418.267,Z 666.157,A -85,B 0,C 180,E1 -10050.893,E2 -10050.893} C_VEL
LIN {X 0,Y 418.261,Z 666.192,A -85,B 0,C 180,E1 -10054.096,E2 -10054.096} C_VEL
LIN {X 0,Y 418.265,Z 666.187,A -85,B 0,C 180,E1 -10057.537,E2 -10057.537} C_VEL
LIN {X 0,Y 418.307,Z 666.188,A -85,B 0,C 180,E1 -10060.366,E2 -10060.366} C_VEL
LIN {X 0,Y 418.306,Z 666.182,A -85,B 0,C 180,E1 -10063.405,E2 -10063.405} C_VEL
LIN {X 0,Y 418.336,Z 666.17,A -85,B 0,C 180,E1 -10066.999,E2 -10066.999} C_VEL
LIN {X 0,Y 418.348,Z 666.183,A -85,B 0,C 180,E1 -10070.329,E2 -10070.329} C_VEL
LIN {X 0,Y 418.485,Z 666.161,A -85,B 0,C 180,E1 -10073.249,E2 -10073.249} C_VEL
LIN {X 0,Y 418.337,Z 666.184,A -85,B 0,C 180,E1 -10075.182,E2 -10075.182} C_VEL
LIN {X 0,Y 418.535,Z 666.148,A -85,B 0,C 180,E1 -10078.076,E2 -10078.076} C_VEL
LIN {X 0,Y 418.664,Z 666.145,A -85,B 0,C 180,E1 -10080,E2 -10080} C_VEL
LIN {X 0,Y 418.502,Z 666.155,A -85,B 0,C 180,E1 -10082.888,E2 -10082.888} C_VEL
LIN {X 0,Y 418.524,Z 666.16,A -85,B 0,C 180,E1 -10085.783,E2 -10085.783} C_VEL
LIN {X 0,Y 418.391,Z 666.166,A -85,B 0,C 180,E1 -10088.695,E2 -10088.695} C_VEL
LIN {X 0,Y 418.327,Z 666.18,A -85,B 0,C 180,E1 -10091.631,E2 -10091.631} C_VEL
LIN {X 0,Y 418.298,Z 666.186,A -85,B 0,C 180,E1 -10094.597,E2 -10094.597} C_VEL
LIN {X 0,Y 418.279,Z 666.183,A -85,B 0,C 180,E1 -10097.604,E2 -10097.604} C_VEL
LIN {X 0,Y 418.251,Z 666.196,A -85,B 0,C 180,E1 -10100.663,E2 -10100.663} C_VEL
LIN {X 0,Y 418.279,Z 666.193,A -85,B 0,C 180,E1 -10103.782,E2 -10103.782} C_VEL
LIN {X 0,Y 418.302,Z 666.169,A -85,B 0,C 180,E1 -10107.071,E2 -10107.071} C_VEL
LIN {X 0,Y 418.253,Z 666.169,A -85,B 0,C 180,E1 -10110.271,E2 -10110.271} C_VEL
LIN {X 0,Y 418.241,Z 666.195,A -85,B 0,C 180,E1 -10113.678,E2 -10113.678} C_VEL
LIN {X 0,Y 418.241,Z 666.19,A -85,B 0,C 180,E1 -10117.224,E2 -10117.224} C_VEL
LIN {X 0,Y 418.261,Z 666.191,A -85,B 0,C 180,E1 -10119.681,E2 -10119.681} C_VEL
LIN {X 0,Y 418.279,Z 666.182,A -85,B 0,C 180,E1 -10122.33,E2 -10122.33} C_VEL
LIN {X 0,Y 418.249,Z 666.181,A -85,B 0,C 180,E1 -10125.112,E2 -10125.112} C_VEL
LIN {X 0,Y 418.237,Z 666.2,A -85,B 0,C 180,E1 -10127.768,E2 -10127.768} C_VEL
LIN {X 0,Y 418.295,Z 666.384,A -85,B 0,C 180,E1 -10131.41,E2 -10131.41} C_VEL
LIN {X 0,Y 422.026,Z 680.332,A -85,B 0,C 180,E1 -10134.686,E2 -10134.686} C_VEL
LIN {X 0,Y 424.863,Z 691.805,A -85,B 0,C 180,E1 -10137.118,E2 -10137.118} C_VEL
LIN {X 0,Y 429.059,Z 701.218,A -85,B 0,C 180,E1 -10137.685,E2 -10137.685} C_VEL
LIN {X 0,Y 435.59,Z 727.817,A -85,B 0,C 180,E1 -10138.725,E2 -10138.725} C_VEL
LIN {X 0,Y 436.564,Z 733.153,A -85,B 0,C 180,E1 -10138.903,E2 -10138.903} C_VEL
LIN {X 0,Y 433.266,Z 894.802,A -85,B 0,C 180,E1 -10141.692,E2 -10141.692} C_VEL
LIN {X 0,Y 432.644,Z 907.272,A -85,B 0,C 180,E1 -10141.995,E2 -10141.995} C_VEL
LIN {X 0,Y 431.872,Z 919.632,A -85,B 0,C 180,E1 -10142.402,E2 -10142.402} C_VEL
LIN {X 0,Y 430.916,Z 932.753,A -85,B 0,C 180,E1 -10142.96,E2 -10142.96} C_VEL
LIN {X 0,Y 429.904,Z 944.141,A -85,B 0,C 180,E1 -10143.547,E2 -10143.547} C_VEL
LIN {X 0,Y 428.648,Z 957.542,A -85,B 0,C 180,E1 -10144.391,E2 -10144.391} C_VEL
LIN {X 0,Y 427.267,Z 970.124,A -85,B 0,C 180,E1 -10145.331,E2 -10145.331} C_VEL
LIN {X 0,Y 426.068,Z 981.127,A -85,B 0,C 180,E1 -10146.293,E2 -10146.293} C_VEL
LIN {X 0,Y 424.743,Z 991.93,A -85,B 0,C 180,E1 -10147.375,E2 -10147.375} C_VEL
LIN {X 0,Y 423.419,Z 1002.432,A -85,B 0,C 180,E1 -10148.583,E2 -10148.583} C_VEL
LIN {X 0,Y 422.281,Z 1011.706,A -85,B 0,C 180,E1 -10149.798,E2 -10149.798} C_VEL
LIN {X 0,Y 421.059,Z 1021.442,A -85,B 0,C 180,E1 -10151.259,E2 -10151.259} C_VEL
LIN {X 0,Y 420.056,Z 1029.968,A -85,B 0,C 180,E1 -10152.724,E2 -10152.724} C_VEL
LIN {X 0,Y 419.107,Z 1038.57,A -85,B 0,C 180,E1 -10154.437,E2 -10154.437} C_VEL
LIN {X 0,Y 418.514,Z 1045.002,A -85,B 0,C 180,E1 -10155.908,E2 -10155.908} C_VEL
LIN {X 0,Y 418.059,Z 1050.641,A -85,B 0,C 180,E1 -10157.377,E2 -10157.377} C_VEL
LIN {X 0,Y 417.545,Z 1056.91,A -85,B 0,C 180,E1 -10159.33,E2 -10159.33} C_VEL
LIN {X 0,Y 417.255,Z 1062.001,A -85,B 0,C 180,E1 -10161.281,E2 -10161.281} C_VEL
LIN {X 0,Y 417.14,Z 1065.994,A -85,B 0,C 180,E1 -10163.227,E2 -10163.227} C_VEL
LIN {X 0,Y 417.043,Z 1068.941,A -85,B 0,C 180,E1 -10165.167,E2 -10165.167} C_VEL
LIN {X 0,Y 416.971,Z 1070.122,A -85,B 0,C 180,E1 -10166.134,E2 -10166.134} C_VEL
LIN {X 0,Y 417.045,Z 1071.587,A -85,B 0,C 180,E1 -10168.069,E2 -10168.069} C_VEL
LIN {X 0,Y 417,Z 1072.07,A -85,B 0,C 180,E1 -10170,E2 -10170} C_VEL
LIN {X 0,Y 417.045,Z 1071.587,A -85,B 0,C 180,E1 -10171.931,E2 -10171.931} C_VEL
LIN {X 0,Y 416.971,Z 1070.122,A -85,B 0,C 180,E1 -10173.866,E2 -10173.866} C_VEL
LIN {X 0,Y 417.14,Z 1066.872,A -85,B 0,C 180,E1 -10176.262,E2 -10176.262} C_VEL
LIN {X 0,Y 417.214,Z 1063.088,A -85,B 0,C 180,E1 -10178.232,E2 -10178.232} C_VEL
LIN {X 0,Y 417.324,Z 1059.602,A -85,B 0,C 180,E1 -10179.695,E2 -10179.695} C_VEL
LIN {X 0,Y 417.741,Z 1053.882,A -85,B 0,C 180,E1 -10181.647,E2 -10181.647} C_VEL
LIN {X 0,Y 418.176,Z 1048.764,A -85,B 0,C 180,E1 -10183.129,E2 -10183.129} C_VEL
LIN {X 0,Y 418.88,Z 1040.793,A -85,B 0,C 180,E1 -10185.073,E2 -10185.073} C_VEL
LIN {X 0,Y 419.722,Z 1033.812,A -85,B 0,C 180,E1 -10186.538,E2 -10186.538} C_VEL
LIN {X 0,Y 420.563,Z 1025.843,A -85,B 0,C 180,E1 -10188.007,E2 -10188.007} C_VEL
LIN {X 0,Y 421.65,Z 1016.724,A -85,B 0,C 180,E1 -10189.472,E2 -10189.472} C_VEL
LIN {X 0,Y 422.714,Z 1008.153,A -85,B 0,C 180,E1 -10190.689,E2 -10190.689} C_VEL
LIN {X 0,Y 424.206,Z 996.069,A -85,B 0,C 180,E1 -10192.167,E2 -10192.167} C_VEL
LIN {X 0,Y 425.472,Z 986.116,A -85,B 0,C 180,E1 -10193.226,E2 -10193.226} C_VEL
LIN {X 0,Y 426.733,Z 974.438,A -85,B 0,C 180,E1 -10194.313,E2 -10194.313} C_VEL
LIN {X 0,Y 428.14,Z 962.411,A -85,B 0,C 180,E1 -10195.264,E2 -10195.264} C_VEL
LIN {X 0,Y 429.383,Z 949.946,A -85,B 0,C 180,E1 -10196.105,E2 -10196.105} C_VEL
LIN {X 0,Y 430.549,Z 937.541,A -85,B 0,C 180,E1 -10196.803,E2 -10196.803} C_VEL
LIN {X 0,Y 431.595,Z 924.111,A -85,B 0,C 180,E1 -10197.42,E2 -10197.42} C_VEL
LIN {X 0,Y 432.355,Z 911.187,A -85,B 0,C 180,E1 -10197.894,E2 -10197.894} C_VEL
LIN {X 0,Y 433.115,Z 898.134,A -85,B 0,C 180,E1 -10198.241,E2 -10198.241} C_VEL
LIN {X 0,Y 433.716,Z 875.624,A -85,B 0,C 180,E1 -10198.66,E2 -10198.66} C_VEL
LIN {X 0,Y 436.507,Z 731.909,A -85,B 0,C 180,E1 -10201.125,E2 -10201.125} C_VEL
LIN {X 0,Y 429.438,Z 702.497,A -85,B 0,C 180,E1 -10202.259,E2 -10202.259} C_VEL
LIN {X 0,Y 427.769,Z 698.244,A -85,B 0,C 180,E1 -10202.481,E2 -10202.481} C_VEL
LIN {X 0,Y 424.843,Z 691.823,A -85,B 0,C 180,E1 -10202.882,E2 -10202.882} C_VEL
LIN {X 0,Y 422.048,Z 680.301,A -85,B 0,C 180,E1 -10205.318,E2 -10205.318} C_VEL
LIN {X 0,Y 418.295,Z 666.364,A -85,B 0,C 180,E1 -10208.59,E2 -10208.59} C_VEL
LIN {X 0,Y 418.227,Z 666.202,A -85,B 0,C 180,E1 -10212.321,E2 -10212.321} C_VEL
LIN {X 0,Y 418.255,Z 666.182,A -85,B 0,C 180,E1 -10215.111,E2 -10215.111} C_VEL
LIN {X 0,Y 418.287,Z 666.18,A -85,B 0,C 180,E1 -10217.773,E2 -10217.773} C_VEL
LIN {X 0,Y 418.261,Z 666.2,A -85,B 0,C 180,E1 -10221.559,E2 -10221.559} C_VEL
LIN {X 0,Y 418.252,Z 666.179,A -85,B 0,C 180,E1 -10225.158,E2 -10225.158} C_VEL
LIN {X 0,Y 418.238,Z 666.199,A -85,B 0,C 180,E1 -10227.471,E2 -10227.471} C_VEL
LIN {X 0,Y 418.268,Z 666.151,A -85,B 0,C 180,E1 -10230.893,E2 -10230.893} C_VEL
LIN {X 0,Y 418.263,Z 666.189,A -85,B 0,C 180,E1 -10234.095,E2 -10234.095} C_VEL
LIN {X 0,Y 418.229,Z 666.187,A -85,B 0,C 180,E1 -10237.263,E2 -10237.263} C_VEL
LIN {X 0,Y 418.307,Z 666.193,A -85,B 0,C 180,E1 -10240.365,E2 -10240.365} C_VEL
LIN {X 0,Y 418.308,Z 666.188,A -85,B 0,C 180,E1 -10243.404,E2 -10243.404} C_VEL
LIN {X 0,Y 418.346,Z 666.175,A -85,B 0,C 180,E1 -10246.993,E2 -10246.993} C_VEL
LIN {X 0,Y 418.352,Z 666.183,A -85,B 0,C 180,E1 -10250.329,E2 -10250.329} C_VEL
LIN {X 0,Y 418.486,Z 666.161,A -85,B 0,C 180,E1 -10253.249,E2 -10253.249} C_VEL
LIN {X 0,Y 418.337,Z 666.186,A -85,B 0,C 180,E1 -10255.181,E2 -10255.181} C_VEL
LIN {X 0,Y 418.535,Z 666.154,A -85,B 0,C 180,E1 -10258.075,E2 -10258.075} C_VEL
LIN {X 0,Y 418.664,Z 666.144,A -85,B 0,C 180,E1 -10260,E2 -10260} C_VEL
LIN {X 0,Y 418.503,Z 666.15,A -85,B 0,C 180,E1 -10262.887,E2 -10262.887} C_VEL
LIN {X 0,Y 418.483,Z 666.162,A -85,B 0,C 180,E1 -10266.596,E2 -10266.596} C_VEL
LIN {X 0,Y 418.348,Z 666.184,A -85,B 0,C 180,E1 -10269.671,E2 -10269.671} C_VEL
LIN {X 0,Y 418.336,Z 666.17,A -85,B 0,C 180,E1 -10273.001,E2 -10273.001} C_VEL
LIN {X 0,Y 418.302,Z 666.182,A -85,B 0,C 180,E1 -10276.735,E2 -10276.735} C_VEL
LIN {X 0,Y 418.294,Z 666.191,A -85,B 0,C 180,E1 -10279.803,E2 -10279.803} C_VEL
LIN {X 0,Y 418.237,Z 666.192,A -85,B 0,C 180,E1 -10282.736,E2 -10282.736} C_VEL
LIN {X 0,Y 418.261,Z 666.192,A -85,B 0,C 180,E1 -10285.904,E2 -10285.904} C_VEL
LIN {X 0,Y 418.264,Z 666.157,A -85,B 0,C 180,E1 -10289.161,E2 -10289.161} C_VEL
LIN {X 0,Y 418.248,Z 666.2,A -85,B 0,C 180,E1 -10292.844,E2 -10292.844} C_VEL
LIN {X 0,Y 418.239,Z 666.164,A -85,B 0,C 180,E1 -10296.239,E2 -10296.239} C_VEL
LIN {X 0,Y 418.258,Z 666.197,A -85,B 0,C 180,E1 -10299.681,E2 -10299.681} C_VEL
LIN {X 0,Y 418.277,Z 666.195,A -85,B 0,C 180,E1 -10302.33,E2 -10302.33} C_VEL
LIN {X 0,Y 418.243,Z 666.202,A -85,B 0,C 180,E1 -10305.111,E2 -10305.111} C_VEL
LIN {X 0,Y 418.248,Z 666.2,A -85,B 0,C 180,E1 -10307.769,E2 -10307.769} C_VEL
LIN {X 0,Y 418.26,Z 666.196,A -85,B 0,C 180,E1 -10310.617,E2 -10310.617} C_VEL
LIN {X 0,Y 418.239,Z 666.2,A -85,B 0,C 180,E1 -10313.977,E2 -10313.977} C_VEL
LIN {X 0,Y 418.251,Z 666.198,A -85,B 0,C 180,E1 -10317.156,E2 -10317.156} C_VEL
LIN {X 0,Y 418.269,Z 666.196,A -85,B 0,C 180,E1 -10320.839,E2 -10320.839} C_VEL
LIN {X 0,Y 418.266,Z 666.197,A -85,B 0,C 180,E1 -10324.096,E2 -10324.096} C_VEL
LIN {X 0,Y 418.233,Z 666.202,A -85,B 0,C 180,E1 -10327.264,E2 -10327.264} C_VEL
LIN {X 0,Y 418.278,Z 666.196,A -85,B 0,C 180,E1 -10330.365,E2 -10330.365} C_VEL
LIN {X 0,Y 418.313,Z 666.19,A -85,B 0,C 180,E1 -10333.405,E2 -10333.405} C_VEL
LIN {X 0,Y 418.342,Z 666.187,A -85,B 0,C 180,E1 -10337,E2 -10337} C_VEL
LIN {X 0,Y 418.337,Z 666.188,A -85,B 0,C 180,E1 -10340.329,E2 -10340.329} C_VEL
LIN {X 0,Y 418.509,Z 666.168,A -85,B 0,C 180,E1 -10342.28,E2 -10342.28} C_VEL
LIN {X 0,Y 418.51,Z 666.166,A -85,B 0,C 180,E1 -10344.217,E2 -10344.217} C_VEL
LIN {X 0,Y 418.541,Z 666.162,A -85,B 0,C 180,E1 -10348.076,E2 -10348.076} C_VEL
LIN {X 0,Y 418.669,Z 666.148,A -85,B 0,C 180,E1 -10350,E2 -10350} C_VEL
LIN {X 0,Y 418.507,Z 666.168,A -85,B 0,C 180,E1 -10352.888,E2 -10352.888} C_VEL
LIN {X 0,Y 418.49,Z 666.171,A -85,B 0,C 180,E1 -10356.751,E2 -10356.751} C_VEL
LIN {X 0,Y 418.354,Z 666.184,A -85,B 0,C 180,E1 -10359.15,E2 -10359.15} C_VEL
LIN {X 0,Y 418.351,Z 666.185,A -85,B 0,C 180,E1 -10362.614,E2 -10362.614} C_VEL
LIN {X 0,Y 418.318,Z 666.19,A -85,B 0,C 180,E1 -10363.34,E2 -10363.34} C_VEL
LIN {X 0,Y 417.625,Z 666.278,A -85,B 0,C 180,E1 -10364.143,E2 -10364.143} C_VEL
LIN {X 0,Y 414.746,Z 666.635,A -85,B 0,C 180,E1 -10365.449,E2 -10365.449} C_VEL
LIN {X 0,Y 412.333,Z 666.934,A -85,B 0,C 180,E1 -10366.503,E2 -10366.503} C_VEL
LIN {X 0,Y 411.312,Z 667.065,A -85,B 0,C 180,E1 -10367.318,E2 -10367.318} C_VEL
LIN {X 0,Y 411.235,Z 667.07,A -85,B 0,C 180,E1 -10367.594,E2 -10367.594} C_VEL
LIN {X 0,Y 411.192,Z 667.078,A -85,B 0,C 180,E1 -10371.034,E2 -10371.034} C_VEL
LIN {X 0,Y 411.222,Z 667.075,A -85,B 0,C 180,E1 -10374.215,E2 -10374.215} C_VEL
LIN {X 0,Y 411.254,Z 667.07,A -85,B 0,C 180,E1 -10377.477,E2 -10377.477} C_VEL
LIN {X 0,Y 411.192,Z 667.079,A -85,B 0,C 180,E1 -10380.846,E2 -10380.846} C_VEL
LIN {X 0,Y 411.199,Z 667.078,A -85,B 0,C 180,E1 -10384.333,E2 -10384.333} C_VEL
LIN {X 0,Y 411.197,Z 667.079,A -85,B 0,C 180,E1 -10387.972,E2 -10387.972} C_VEL
LIN {X 0,Y 411.193,Z 667.078,A -85,B 0,C 180,E1 -10391.234,E2 -10391.234} C_VEL
LIN {X 0,Y 411.176,Z 667.082,A -85,B 0,C 180,E1 -10394.489,E2 -10394.489} C_VEL
LIN {X 0,Y 411.223,Z 667.075,A -85,B 0,C 180,E1 -10397.296,E2 -10397.296} C_VEL
LIN {X 0,Y 411.223,Z 667.076,A -85,B 0,C 180,E1 -10400.777,E2 -10400.777} C_VEL
LIN {X 0,Y 411.19,Z 667.044,A -85,B 0,C 180,E1 -10404.471,E2 -10404.471} C_VEL
LIN {X 0,Y 411.198,Z 667.075,A -85,B 0,C 180,E1 -10406.873,E2 -10406.873} C_VEL
LIN {X 0,Y 411.231,Z 667.033,A -85,B 0,C 180,E1 -10410.642,E2 -10410.642} C_VEL
LIN {X 0,Y 411.228,Z 667.058,A -85,B 0,C 180,E1 -10413.619,E2 -10413.619} C_VEL
LIN {X 0,Y 411.199,Z 667.071,A -85,B 0,C 180,E1 -10416.853,E2 -10416.853} C_VEL
LIN {X 0,Y 411.255,Z 667.07,A -85,B 0,C 180,E1 -10420.031,E2 -10420.031} C_VEL
LIN {X 0,Y 411.253,Z 667.059,A -85,B 0,C 180,E1 -10423.131,E2 -10423.131} C_VEL
LIN {X 0,Y 411.295,Z 667.047,A -85,B 0,C 180,E1 -10426.896,E2 -10426.896} C_VEL
LIN {X 0,Y 411.295,Z 667.064,A -85,B 0,C 180,E1 -10430.162,E2 -10430.162} C_VEL
LIN {X 0,Y 411.448,Z 667.037,A -85,B 0,C 180,E1 -10433.133,E2 -10433.133} C_VEL
LIN {X 0,Y 411.309,Z 667.06,A -85,B 0,C 180,E1 -10435.099,E2 -10435.099} C_VEL
LIN {X 0,Y 411.504,Z 667.023,A -85,B 0,C 180,E1 -10438.043,E2 -10438.043} C_VEL
LIN {X 0,Y 411.633,Z 667.021,A -85,B 0,C 180,E1 -10440,E2 -10440} C_VEL
LIN {X 0,Y 411.458,Z 667.032,A -85,B 0,C 180,E1 -10442.937,E2 -10442.937} C_VEL
LIN {X 0,Y 411.483,Z 667.037,A -85,B 0,C 180,E1 -10445.882,E2 -10445.882} C_VEL
LIN {X 0,Y 411.348,Z 667.044,A -85,B 0,C 180,E1 -10448.846,E2 -10448.846} C_VEL
LIN {X 0,Y 411.293,Z 667.055,A -85,B 0,C 180,E1 -10451.833,E2 -10451.833} C_VEL
LIN {X 0,Y 411.254,Z 667.065,A -85,B 0,C 180,E1 -10454.853,E2 -10454.853} C_VEL
LIN {X 0,Y 411.243,Z 667.059,A -85,B 0,C 180,E1 -10457.916,E2 -10457.916} C_VEL
LIN {X 0,Y 411.193,Z 667.077,A -85,B 0,C 180,E1 -10461.034,E2 -10461.034} C_VEL
LIN {X 0,Y 411.219,Z 667.074,A -85,B 0,C 180,E1 -10464.216,E2 -10464.216} C_VEL
LIN {X 0,Y 411.252,Z 667.036,A -85,B 0,C 180,E1 -10467.478,E2 -10467.478} C_VEL
LIN {X 0,Y 411.19,Z 667.063,A -85,B 0,C 180,E1 -10470.848,E2 -10470.848} C_VEL
LIN {X 0,Y 411.199,Z 667.061,A -85,B 0,C 180,E1 -10474.334,E2 -10474.334} C_VEL
LIN {X 0,Y 411.199,Z 667.073,A -85,B 0,C 180,E1 -10477.973,E2 -10477.973} C_VEL
LIN {X 0,Y 411.204,Z 667.053,A -85,B 0,C 180,E1 -10481.236,E2 -10481.236} C_VEL
LIN {X 0,Y 411.224,Z 667.062,A -85,B 0,C 180,E1 -10484.484,E2 -10484.484} C_VEL
LIN {X 0,Y 411.174,Z 667.072,A -85,B 0,C 180,E1 -10488.196,E2 -10488.196} C_VEL
LIN {X 0,Y 411.242,Z 667.264,A -85,B 0,C 180,E1 -10490.867,E2 -10490.867} C_VEL
LIN {X 0,Y 414.862,Z 680.622,A -85,B 0,C 180,E1 -10494.092,E2 -10494.092} C_VEL
LIN {X 0,Y 417.614,Z 691.548,A -85,B 0,C 180,E1 -10496.474,E2 -10496.474} C_VEL
LIN {X 0,Y 423.52,Z 704.581,A -85,B 0,C 180,E1 -10497.28,E2 -10497.28} C_VEL
LIN {X 0,Y 429.752,Z 730.337,A -85,B 0,C 180,E1 -10498.304,E2 -10498.304} C_VEL
LIN {X 0,Y 430.431,Z 733.399,A -85,B 0,C 180,E1 -10498.418,E2 -10498.418} C_VEL
LIN {X 0,Y 427.211,Z 888.899,A -85,B 0,C 180,E1 -10501.118,E2 -10501.118} C_VEL
LIN {X 0,Y 426.495,Z 905.108,A -85,B 0,C 180,E1 -10501.488,E2 -10501.488} C_VEL
LIN {X 0,Y 425.569,Z 918.677,A -85,B 0,C 180,E1 -10501.924,E2 -10501.924} C_VEL
LIN {X 0,Y 424.582,Z 932.547,A -85,B 0,C 180,E1 -10502.523,E2 -10502.523} C_VEL
LIN {X 0,Y 423.538,Z 943.935,A -85,B 0,C 180,E1 -10503.118,E2 -10503.118} C_VEL
LIN {X 0,Y 422.26,Z 957.047,A -85,B 0,C 180,E1 -10503.952,E2 -10503.952} C_VEL
LIN {X 0,Y 420.79,Z 969.917,A -85,B 0,C 180,E1 -10504.925,E2 -10504.925} C_VEL
LIN {X 0,Y 419.441,Z 980.917,A -85,B 0,C 180,E1 -10505.895,E2 -10505.895} C_VEL
LIN {X 0,Y 418.125,Z 991.722,A -85,B 0,C 180,E1 -10506.997,E2 -10506.997} C_VEL
LIN {X 0,Y 416.722,Z 1002.224,A -85,B 0,C 180,E1 -10508.222,E2 -10508.222} C_VEL
LIN {X 0,Y 415.516,Z 1011.498,A -85,B 0,C 180,E1 -10509.454,E2 -10509.454} C_VEL
LIN {X 0,Y 414.227,Z 1021.233,A -85,B 0,C 180,E1 -10510.938,E2 -10510.938} C_VEL
LIN {X 0,Y 413.202,Z 1029.598,A -85,B 0,C 180,E1 -10512.396,E2 -10512.396} C_VEL
LIN {X 0,Y 412.336,Z 1037.251,A -85,B 0,C 180,E1 -10513.921,E2 -10513.921} C_VEL
LIN {X 0,Y 411.524,Z 1044.794,A -85,B 0,C 180,E1 -10515.663,E2 -10515.663} C_VEL
LIN {X 0,Y 411.014,Z 1050.432,A -85,B 0,C 180,E1 -10517.157,E2 -10517.157} C_VEL
LIN {X 0,Y 410.485,Z 1056.702,A -85,B 0,C 180,E1 -10519.145,E2 -10519.145} C_VEL
LIN {X 0,Y 410.189,Z 1061.795,A -85,B 0,C 180,E1 -10521.13,E2 -10521.13} C_VEL
LIN {X 0,Y 410.048,Z 1065.787,A -85,B 0,C 180,E1 -10523.109,E2 -10523.109} C_VEL
LIN {X 0,Y 409.954,Z 1068.735,A -85,B 0,C 180,E1 -10525.083,E2 -10525.083} C_VEL
LIN {X 0,Y 409.889,Z 1069.917,A -85,B 0,C 180,E1 -10526.067,E2 -10526.067} C_VEL
LIN {X 0,Y 409.955,Z 1071.381,A -85,B 0,C 180,E1 -10528.035,E2 -10528.035} C_VEL
LIN {X 0,Y 409.922,Z 1071.865,A -85,B 0,C 180,E1 -10530,E2 -10530} C_VEL
LIN {X 0,Y 409.955,Z 1071.381,A -85,B 0,C 180,E1 -10531.965,E2 -10531.965} C_VEL
LIN {X 0,Y 409.889,Z 1069.917,A -85,B 0,C 180,E1 -10533.933,E2 -10533.933} C_VEL
LIN {X 0,Y 410.04,Z 1066.914,A -85,B 0,C 180,E1 -10536.225,E2 -10536.225} C_VEL
LIN {X 0,Y 410.128,Z 1062.881,A -85,B 0,C 180,E1 -10538.375,E2 -10538.375} C_VEL
LIN {X 0,Y 410.256,Z 1059.395,A -85,B 0,C 180,E1 -10539.864,E2 -10539.864} C_VEL
LIN {X 0,Y 410.708,Z 1053.674,A -85,B 0,C 180,E1 -10541.849,E2 -10541.849} C_VEL
LIN {X 0,Y 411.244,Z 1047.757,A -85,B 0,C 180,E1 -10543.565,E2 -10543.565} C_VEL
LIN {X 0,Y 411.919,Z 1040.584,A -85,B 0,C 180,E1 -10545.334,E2 -10545.334} C_VEL
LIN {X 0,Y 412.808,Z 1033.603,A -85,B 0,C 180,E1 -10546.823,E2 -10546.823} C_VEL
LIN {X 0,Y 413.705,Z 1025.631,A -85,B 0,C 180,E1 -10548.317,E2 -10548.317} C_VEL
LIN {X 0,Y 414.854,Z 1016.515,A -85,B 0,C 180,E1 -10549.804,E2 -10549.804} C_VEL
LIN {X 0,Y 415.979,Z 1007.944,A -85,B 0,C 180,E1 -10551.039,E2 -10551.039} C_VEL
LIN {X 0,Y 417.522,Z 996.093,A -85,B 0,C 180,E1 -10552.513,E2 -10552.513} C_VEL
LIN {X 0,Y 418.874,Z 985.908,A -85,B 0,C 180,E1 -10553.614,E2 -10553.614} C_VEL
LIN {X 0,Y 420.214,Z 974.231,A -85,B 0,C 180,E1 -10554.715,E2 -10554.715} C_VEL
LIN {X 0,Y 421.679,Z 962.204,A -85,B 0,C 180,E1 -10555.679,E2 -10555.679} C_VEL
LIN {X 0,Y 422.97,Z 949.728,A -85,B 0,C 180,E1 -10556.532,E2 -10556.532} C_VEL
LIN {X 0,Y 424.208,Z 937.335,A -85,B 0,C 180,E1 -10557.236,E2 -10557.236} C_VEL
LIN {X 0,Y 425.261,Z 923.904,A -85,B 0,C 180,E1 -10557.864,E2 -10557.864} C_VEL
LIN {X 0,Y 426.095,Z 910.982,A -85,B 0,C 180,E1 -10558.34,E2 -10558.34} C_VEL
LIN {X 0,Y 426.855,Z 898.195,A -85,B 0,C 180,E1 -10558.686,E2 -10558.686} C_VEL
LIN {X 0,Y 427.483,Z 875.408,A -85,B 0,C 180,E1 -10559.118,E2 -10559.118} C_VEL
LIN {X 0,Y 430.451,Z 733.465,A -85,B 0,C 180,E1 -10561.579,E2 -10561.579} C_VEL
LIN {X 0,Y 423.522,Z 704.433,A -85,B 0,C 180,E1 -10562.723,E2 -10562.723} C_VEL
LIN {X 0,Y 417.592,Z 691.626,A -85,B 0,C 180,E1 -10563.521,E2 -10563.521} C_VEL
LIN {X 0,Y 415.854,Z 684.28,A -85,B 0,C 180,E1 -10565.071,E2 -10565.071} C_VEL
LIN {X 0,Y 412.087,Z 670.439,A -85,B 0,C 180,E1 -10568.324,E2 -10568.324} C_VEL
LIN {X 0,Y 411.215,Z 667.099,A -85,B 0,C 180,E1 -10569.206,E2 -10569.206} C_VEL
LIN {X 0,Y 411.18,Z 667.081,A -85,B 0,C 180,E1 -10572.696,E2 -10572.696} C_VEL
LIN {X 0,Y 411.231,Z 667.068,A -85,B 0,C 180,E1 -10575.87,E2 -10575.87} C_VEL
LIN {X 0,Y 411.204,Z 667.053,A -85,B 0,C 180,E1 -10578.764,E2 -10578.764} C_VEL
LIN {X 0,Y 411.199,Z 667.073,A -85,B 0,C 180,E1 -10582.027,E2 -10582.027} C_VEL
LIN {X 0,Y 411.199,Z 667.061,A -85,B 0,C 180,E1 -10585.666,E2 -10585.666} C_VEL
LIN {X 0,Y 411.19,Z 667.063,A -85,B 0,C 180,E1 -10589.152,E2 -10589.152} C_VEL
LIN {X 0,Y 411.252,Z 667.036,A -85,B 0,C 180,E1 -10592.522,E2 -10592.522} C_VEL
LIN {X 0,Y 411.219,Z 667.074,A -85,B 0,C 180,E1 -10595.784,E2 -10595.784} C_VEL
LIN {X 0,Y 411.193,Z 667.077,A -85,B 0,C 180,E1 -10598.966,E2 -10598.966} C_VEL
LIN {X 0,Y 411.243,Z 667.059,A -85,B 0,C 180,E1 -10602.084,E2 -10602.084} C_VEL
LIN {X 0,Y 411.254,Z 667.067,A -85,B 0,C 180,E1 -10605.147,E2 -10605.147} C_VEL
LIN {X 0,Y 411.293,Z 667.056,A -85,B 0,C 180,E1 -10608.167,E2 -10608.167} C_VEL
LIN {X 0,Y 411.434,Z 667.029,A -85,B 0,C 180,E1 -10612.185,E2 -10612.185} C_VEL
LIN {X 0,Y 411.483,Z 667.036,A -85,B 0,C 180,E1 -10614.118,E2 -10614.118} C_VEL
LIN {X 0,Y 411.504,Z 667.03,A -85,B 0,C 180,E1 -10618.042,E2 -10618.042} C_VEL
LIN {X 0,Y 411.633,Z 667.02,A -85,B 0,C 180,E1 -10620,E2 -10620} C_VEL
LIN {X 0,Y 411.458,Z 667.028,A -85,B 0,C 180,E1 -10622.937,E2 -10622.937} C_VEL
LIN {X 0,Y 411.445,Z 667.038,A -85,B 0,C 180,E1 -10626.595,E2 -10626.595} C_VEL
LIN {X 0,Y 411.295,Z 667.065,A -85,B 0,C 180,E1 -10629.838,E2 -10629.838} C_VEL
LIN {X 0,Y 411.295,Z 667.047,A -85,B 0,C 180,E1 -10633.104,E2 -10633.104} C_VEL
LIN {X 0,Y 411.247,Z 667.06,A -85,B 0,C 180,E1 -10636.889,E2 -10636.889} C_VEL
LIN {X 0,Y 411.246,Z 667.072,A -85,B 0,C 180,E1 -10639.986,E2 -10639.986} C_VEL
LIN {X 0,Y 411.199,Z 667.071,A -85,B 0,C 180,E1 -10643.147,E2 -10643.147} C_VEL
LIN {X 0,Y 411.228,Z 667.057,A -85,B 0,C 180,E1 -10646.381,E2 -10646.381} C_VEL
LIN {X 0,Y 411.201,Z 667.042,A -85,B 0,C 180,E1 -10649.712,E2 -10649.712} C_VEL
LIN {X 0,Y 411.197,Z 667.074,A -85,B 0,C 180,E1 -10653.156,E2 -10653.156} C_VEL
LIN {X 0,Y 411.187,Z 667.043,A -85,B 0,C 180,E1 -10656.553,E2 -10656.553} C_VEL
LIN {X 0,Y 411.22,Z 667.073,A -85,B 0,C 180,E1 -10659.731,E2 -10659.731} C_VEL
LIN {X 0,Y 411.22,Z 667.077,A -85,B 0,C 180,E1 -10663.127,E2 -10663.127} C_VEL
LIN {X 0,Y 411.164,Z 667.081,A -85,B 0,C 180,E1 -10665.881,E2 -10665.881} C_VEL
LIN {X 0,Y 411.204,Z 667.078,A -85,B 0,C 180,E1 -10669.5,E2 -10669.5} C_VEL
LIN {X 0,Y 411.197,Z 667.078,A -85,B 0,C 180,E1 -10672.028,E2 -10672.028} C_VEL
LIN {X 0,Y 411.199,Z 667.078,A -85,B 0,C 180,E1 -10675.667,E2 -10675.667} C_VEL
LIN {X 0,Y 411.192,Z 667.079,A -85,B 0,C 180,E1 -10679.154,E2 -10679.154} C_VEL
LIN {X 0,Y 411.254,Z 667.069,A -85,B 0,C 180,E1 -10682.523,E2 -10682.523} C_VEL
LIN {X 0,Y 411.222,Z 667.075,A -85,B 0,C 180,E1 -10685.785,E2 -10685.785} C_VEL
LIN {X 0,Y 411.192,Z 667.078,A -85,B 0,C 180,E1 -10688.966,E2 -10688.966} C_VEL
LIN {X 0,Y 411.248,Z 667.071,A -85,B 0,C 180,E1 -10692.085,E2 -10692.085} C_VEL
LIN {X 0,Y 411.255,Z 667.071,A -85,B 0,C 180,E1 -10695.148,E2 -10695.148} C_VEL
LIN {X 0,Y 411.28,Z 667.069,A -85,B 0,C 180,E1 -10698.167,E2 -10698.167} C_VEL
LIN {X 0,Y 411.478,Z 667.044,A -85,B 0,C 180,E1 -10702.147,E2 -10702.147} C_VEL
LIN {X 0,Y 411.472,Z 667.043,A -85,B 0,C 180,E1 -10704.118,E2 -10704.118} C_VEL
LIN {X 0,Y 411.51,Z 667.038,A -85,B 0,C 180,E1 -10708.043,E2 -10708.043} C_VEL
LIN {X 0,Y 411.639,Z 667.025,A -85,B 0,C 180,E1 -10710,E2 -10710} C_VEL
LIN {X 0,Y 411.463,Z 667.045,A -85,B 0,C 180,E1 -10712.937,E2 -10712.937} C_VEL
LIN {X 0,Y 411.457,Z 667.046,A -85,B 0,C 180,E1 -10716.867,E2 -10716.867} C_VEL
LIN {X 0,Y 411.289,Z 667.066,A -85,B 0,C 180,E1 -10719.839,E2 -10719.839} C_VEL
LIN {X 0,Y 411.278,Z 667.067,A -85,B 0,C 180,E1 -10723.328,E2 -10723.328} C_VEL
LIN {X 0,Y 411.253,Z 667.07,A -85,B 0,C 180,E1 -10726.888,E2 -10726.888} C_VEL
LIN {X 0,Y 411.235,Z 667.07,A -85,B 0,C 180,E1 -10727.594,E2 -10727.594} C_VEL
LIN {X 0,Y 410.575,Z 667.156,A -85,B 0,C 180,E1 -10728.412,E2 -10728.412} C_VEL
LIN {X 0,Y 407.687,Z 667.517,A -85,B 0,C 180,E1 -10729.74,E2 -10729.74} C_VEL
LIN {X 0,Y 405.243,Z 667.821,A -85,B 0,C 180,E1 -10730.813,E2 -10730.813} C_VEL
LIN {X 0,Y 404.207,Z 667.949,A -85,B 0,C 180,E1 -10731.643,E2 -10731.643} C_VEL
LIN {X 0,Y 404.131,Z 667.958,A -85,B 0,C 180,E1 -10731.924,E2 -10731.924} C_VEL
LIN {X 0,Y 404.211,Z 667.949,A -85,B 0,C 180,E1 -10735.296,E2 -10735.296} C_VEL
LIN {X 0,Y 404.192,Z 667.952,A -85,B 0,C 180,E1 -10737.999,E2 -10737.999} C_VEL
LIN {X 0,Y 404.137,Z 667.956,A -85,B 0,C 180,E1 -10741.558,E2 -10741.558} C_VEL
LIN {X 0,Y 404.179,Z 667.952,A -85,B 0,C 180,E1 -10745.016,E2 -10745.016} C_VEL
LIN {X 0,Y 404.156,Z 667.956,A -85,B 0,C 180,E1 -10748.755,E2 -10748.755} C_VEL
LIN {X 0,Y 404.142,Z 667.956,A -85,B 0,C 180,E1 -10751.604,E2 -10751.604} C_VEL
LIN {X 0,Y 404.145,Z 667.958,A -85,B 0,C 180,E1 -10754.523,E2 -10754.523} C_VEL
LIN {X 0,Y 404.201,Z 667.95,A -85,B 0,C 180,E1 -10757.305,E2 -10757.305} C_VEL
LIN {X 0,Y 404.16,Z 667.952,A -85,B 0,C 180,E1 -10759.955,E2 -10759.955} C_VEL
LIN {X 0,Y 404.131,Z 667.923,A -85,B 0,C 180,E1 -10763.124,E2 -10763.124} C_VEL
LIN {X 0,Y 404.136,Z 667.952,A -85,B 0,C 180,E1 -10766.187,E2 -10766.187} C_VEL
LIN {X 0,Y 404.144,Z 667.929,A -85,B 0,C 180,E1 -10769.715,E2 -10769.715} C_VEL
LIN {X 0,Y 404.186,Z 667.928,A -85,B 0,C 180,E1 -10773.123,E2 -10773.123} C_VEL
LIN {X 0,Y 404.163,Z 667.948,A -85,B 0,C 180,E1 -10776.426,E2 -10776.426} C_VEL
LIN {X 0,Y 404.217,Z 667.949,A -85,B 0,C 180,E1 -10779.86,E2 -10779.86} C_VEL
LIN {X 0,Y 404.206,Z 667.936,A -85,B 0,C 180,E1 -10782.993,E2 -10782.993} C_VEL
LIN {X 0,Y 404.273,Z 667.921,A -85,B 0,C 180,E1 -10786.939,E2 -10786.939} C_VEL
LIN {X 0,Y 404.257,Z 667.941,A -85,B 0,C 180,E1 -10789.989,E2 -10789.989} C_VEL
LIN {X 0,Y 404.392,Z 667.915,A -85,B 0,C 180,E1 -10793.013,E2 -10793.013} C_VEL
LIN {X 0,Y 404.281,Z 667.936,A -85,B 0,C 180,E1 -10795.014,E2 -10795.014} C_VEL
LIN {X 0,Y 404.473,Z 667.898,A -85,B 0,C 180,E1 -10798.009,E2 -10798.009} C_VEL
LIN {X 0,Y 404.603,Z 667.897,A -85,B 0,C 180,E1 -10800,E2 -10800} C_VEL
LIN {X 0,Y 404.415,Z 667.909,A -85,B 0,C 180,E1 -10802.989,E2 -10802.989} C_VEL
LIN {X 0,Y 404.429,Z 667.916,A -85,B 0,C 180,E1 -10805.985,E2 -10805.985} C_VEL
LIN {X 0,Y 404.287,Z 667.926,A -85,B 0,C 180,E1 -10809.001,E2 -10809.001} C_VEL
LIN {X 0,Y 404.263,Z 667.93,A -85,B 0,C 180,E1 -10812.041,E2 -10812.041} C_VEL
LIN {X 0,Y 404.199,Z 667.947,A -85,B 0,C 180,E1 -10815.118,E2 -10815.118} C_VEL
LIN {X 0,Y 404.204,Z 667.936,A -85,B 0,C 180,E1 -10818.238,E2 -10818.238} C_VEL
LIN {X 0,Y 404.133,Z 667.951,A -85,B 0,C 180,E1 -10821.42,E2 -10821.42} C_VEL
LIN {X 0,Y 404.169,Z 667.951,A -85,B 0,C 180,E1 -10824.666,E2 -10824.666} C_VEL
LIN {X 0,Y 404.19,Z 667.906,A -85,B 0,C 180,E1 -10828,E2 -10828} C_VEL
LIN {X 0,Y 404.135,Z 667.949,A -85,B 0,C 180,E1 -10831.56,E2 -10831.56} C_VEL
LIN {X 0,Y 404.178,Z 667.927,A -85,B 0,C 180,E1 -10835.017,E2 -10835.017} C_VEL
LIN {X 0,Y 404.159,Z 667.954,A -85,B 0,C 180,E1 -10838.756,E2 -10838.756} C_VEL
LIN {X 0,Y 404.186,Z 667.928,A -85,B 0,C 180,E1 -10841.611,E2 -10841.611} C_VEL
LIN {X 0,Y 404.188,Z 667.938,A -85,B 0,C 180,E1 -10844.53,E2 -10844.53} C_VEL
LIN {X 0,Y 404.134,Z 667.959,A -85,B 0,C 180,E1 -10847.297,E2 -10847.297} C_VEL
LIN {X 0,Y 404.19,Z 668.083,A -85,B 0,C 180,E1 -10850.267,E2 -10850.267} C_VEL
LIN {X 0,Y 407.113,Z 678.856,A -85,B 0,C 180,E1 -10852.978,E2 -10852.978} C_VEL
LIN {X 0,Y 410.242,Z 690.935,A -85,B 0,C 180,E1 -10855.749,E2 -10855.749} C_VEL
LIN {X 0,Y 411.48,Z 693.909,A -85,B 0,C 180,E1 -10855.985,E2 -10855.985} C_VEL
LIN {X 0,Y 417.749,Z 706.943,A -85,B 0,C 180,E1 -10856.821,E2 -10856.821} C_VEL
LIN {X 0,Y 424.355,Z 734.806,A -85,B 0,C 180,E1 -10857.944,E2 -10857.944} C_VEL
LIN {X 0,Y 421.295,Z 875.079,A -85,B 0,C 180,E1 -10860.41,E2 -10860.41} C_VEL
LIN {X 0,Y 420.637,Z 899.182,A -85,B 0,C 180,E1 -10860.878,E2 -10860.878} C_VEL
LIN {X 0,Y 419.353,Z 917.725,A -85,B 0,C 180,E1 -10861.436,E2 -10861.436} C_VEL
LIN {X 0,Y 418.282,Z 932.341,A -85,B 0,C 180,E1 -10862.073,E2 -10862.073} C_VEL
LIN {X 0,Y 417.196,Z 943.729,A -85,B 0,C 180,E1 -10862.675,E2 -10862.675} C_VEL
LIN {X 0,Y 415.921,Z 955.963,A -85,B 0,C 180,E1 -10863.453,E2 -10863.453} C_VEL
LIN {X 0,Y 414.526,Z 968.272,A -85,B 0,C 180,E1 -10864.385,E2 -10864.385} C_VEL
LIN {X 0,Y 412.879,Z 980.708,A -85,B 0,C 180,E1 -10865.487,E2 -10865.487} C_VEL
LIN {X 0,Y 411.494,Z 991.514,A -85,B 0,C 180,E1 -10866.604,E2 -10866.604} C_VEL
LIN {X 0,Y 410.061,Z 1002.016,A -85,B 0,C 180,E1 -10867.849,E2 -10867.849} C_VEL
LIN {X 0,Y 408.761,Z 1011.289,A -85,B 0,C 180,E1 -10869.099,E2 -10869.099} C_VEL
LIN {X 0,Y 407.415,Z 1021.024,A -85,B 0,C 180,E1 -10870.606,E2 -10870.606} C_VEL
LIN {X 0,Y 406.258,Z 1029.984,A -85,B 0,C 180,E1 -10872.206,E2 -10872.206} C_VEL
LIN {X 0,Y 405.248,Z 1038.153,A -85,B 0,C 180,E1 -10873.891,E2 -10873.891} C_VEL
LIN {X 0,Y 404.538,Z 1044.585,A -85,B 0,C 180,E1 -10875.41,E2 -10875.41} C_VEL
LIN {X 0,Y 403.862,Z 1051.89,A -85,B 0,C 180,E1 -10877.45,E2 -10877.45} C_VEL
LIN {X 0,Y 403.44,Z 1056.494,A -85,B 0,C 180,E1 -10878.953,E2 -10878.953} C_VEL
LIN {X 0,Y 403.112,Z 1061.587,A -85,B 0,C 180,E1 -10880.973,E2 -10880.973} C_VEL
LIN {X 0,Y 402.969,Z 1065.581,A -85,B 0,C 180,E1 -10882.988,E2 -10882.988} C_VEL
LIN {X 0,Y 402.916,Z 1067.252,A -85,B 0,C 180,E1 -10883.993,E2 -10883.993} C_VEL
LIN {X 0,Y 402.81,Z 1069.711,A -85,B 0,C 180,E1 -10885.998,E2 -10885.998} C_VEL
LIN {X 0,Y 402.853,Z 1071.176,A -85,B 0,C 180,E1 -10888.001,E2 -10888.001} C_VEL
LIN {X 0,Y 402.847,Z 1071.661,A -85,B 0,C 180,E1 -10890,E2 -10890} C_VEL
LIN {X 0,Y 402.853,Z 1071.176,A -85,B 0,C 180,E1 -10891.999,E2 -10891.999} C_VEL
LIN {X 0,Y 402.81,Z 1069.711,A -85,B 0,C 180,E1 -10894.002,E2 -10894.002} C_VEL
LIN {X 0,Y 402.938,Z 1066.961,A -85,B 0,C 180,E1 -10896.182,E2 -10896.182} C_VEL
LIN {X 0,Y 403.061,Z 1062.674,A -85,B 0,C 180,E1 -10898.523,E2 -10898.523} C_VEL
LIN {X 0,Y 403.191,Z 1059.187,A -85,B 0,C 180,E1 -10900.038,E2 -10900.038} C_VEL
LIN {X 0,Y 403.688,Z 1053.466,A -85,B 0,C 180,E1 -10902.058,E2 -10902.058} C_VEL
LIN {X 0,Y 404.174,Z 1048.408,A -85,B 0,C 180,E1 -10903.576,E2 -10903.576} C_VEL
LIN {X 0,Y 404.967,Z 1040.375,A -85,B 0,C 180,E1 -10905.604,E2 -10905.604} C_VEL
LIN {X 0,Y 405.901,Z 1033.394,A -85,B 0,C 180,E1 -10907.118,E2 -10907.118} C_VEL
LIN {X 0,Y 406.831,Z 1025.421,A -85,B 0,C 180,E1 -10908.637,E2 -10908.637} C_VEL
LIN {X 0,Y 408.057,Z 1016.306,A -85,B 0,C 180,E1 -10910.148,E2 -10910.148} C_VEL
LIN {X 0,Y 409.277,Z 1007.736,A -85,B 0,C 180,E1 -10911.401,E2 -10911.401} C_VEL
LIN {X 0,Y 410.853,Z 995.868,A -85,B 0,C 180,E1 -10912.901,E2 -10912.901} C_VEL
LIN {X 0,Y 412.452,Z 984.452,A -85,B 0,C 180,E1 -10914.138,E2 -10914.138} C_VEL
LIN {X 0,Y 413.711,Z 974.024,A -85,B 0,C 180,E1 -10915.13,E2 -10915.13} C_VEL
LIN {X 0,Y 415.252,Z 961.997,A -85,B 0,C 180,E1 -10916.106,E2 -10916.106} C_VEL
LIN {X 0,Y 416.579,Z 949.661,A -85,B 0,C 180,E1 -10916.962,E2 -10916.962} C_VEL
LIN {X 0,Y 417.854,Z 937.128,A -85,B 0,C 180,E1 -10917.686,E2 -10917.686} C_VEL
LIN {X 0,Y 418.941,Z 923.696,A -85,B 0,C 180,E1 -10918.322,E2 -10918.322} C_VEL
LIN {X 0,Y 419.849,Z 910.776,A -85,B 0,C 180,E1 -10918.801,E2 -10918.801} C_VEL
LIN {X 0,Y 420.697,Z 897.298,A -85,B 0,C 180,E1 -10919.163,E2 -10919.163} C_VEL
LIN {X 0,Y 421.381,Z 872.092,A -85,B 0,C 180,E1 -10919.64,E2 -10919.64} C_VEL
LIN {X 0,Y 424.361,Z 734.724,A -85,B 0,C 180,E1 -10922.058,E2 -10922.058} C_VEL
LIN {X 0,Y 417.903,Z 707.4,A -85,B 0,C 180,E1 -10923.156,E2 -10923.156} C_VEL
LIN {X 0,Y 410.339,Z 691.273,A -85,B 0,C 180,E1 -10924.201,E2 -10924.201} C_VEL
LIN {X 0,Y 408.27,Z 683.167,A -85,B 0,C 180,E1 -10925.996,E2 -10925.996} C_VEL
LIN {X 0,Y 405.033,Z 671.182,A -85,B 0,C 180,E1 -10928.899,E2 -10928.899} C_VEL
LIN {X 0,Y 404.17,Z 667.988,A -85,B 0,C 180,E1 -10929.761,E2 -10929.761} C_VEL
LIN {X 0,Y 404.151,Z 667.95,A -85,B 0,C 180,E1 -10933.083,E2 -10933.083} C_VEL
LIN {X 0,Y 404.204,Z 667.944,A -85,B 0,C 180,E1 -10935.934,E2 -10935.934} C_VEL
LIN {X 0,Y 404.158,Z 667.93,A -85,B 0,C 180,E1 -10938.64,E2 -10938.64} C_VEL
LIN {X 0,Y 404.157,Z 667.956,A -85,B 0,C 180,E1 -10941.49,E2 -10941.49} C_VEL
LIN {X 0,Y 404.178,Z 667.927,A -85,B 0,C 180,E1 -10944.983,E2 -10944.983} C_VEL
LIN {X 0,Y 404.138,Z 667.947,A -85,B 0,C 180,E1 -10948.553,E2 -10948.553} C_VEL
LIN {X 0,Y 404.19,Z 667.906,A -85,B 0,C 180,E1 -10952,E2 -10952} C_VEL
LIN {X 0,Y 404.169,Z 667.951,A -85,B 0,C 180,E1 -10955.334,E2 -10955.334} C_VEL
LIN {X 0,Y 404.133,Z 667.951,A -85,B 0,C 180,E1 -10958.58,E2 -10958.58} C_VEL
LIN {X 0,Y 404.204,Z 667.937,A -85,B 0,C 180,E1 -10961.762,E2 -10961.762} C_VEL
LIN {X 0,Y 404.199,Z 667.949,A -85,B 0,C 180,E1 -10964.882,E2 -10964.882} C_VEL
LIN {X 0,Y 404.263,Z 667.931,A -85,B 0,C 180,E1 -10967.959,E2 -10967.959} C_VEL
LIN {X 0,Y 404.375,Z 667.908,A -85,B 0,C 180,E1 -10972.008,E2 -10972.008} C_VEL
LIN {X 0,Y 404.429,Z 667.915,A -85,B 0,C 180,E1 -10974.015,E2 -10974.015} C_VEL
LIN {X 0,Y 404.473,Z 667.905,A -85,B 0,C 180,E1 -10978.008,E2 -10978.008} C_VEL
LIN {X 0,Y 404.603,Z 667.896,A -85,B 0,C 180,E1 -10980,E2 -10980} C_VEL
LIN {X 0,Y 404.416,Z 667.905,A -85,B 0,C 180,E1 -10982.988,E2 -10982.988} C_VEL
LIN {X 0,Y 404.391,Z 667.916,A -85,B 0,C 180,E1 -10986.592,E2 -10986.592} C_VEL
LIN {X 0,Y 404.285,Z 667.929,A -85,B 0,C 180,E1 -10989.001,E2 -10989.001} C_VEL
LIN {X 0,Y 404.247,Z 667.929,A -85,B 0,C 180,E1 -10992.041,E2 -10992.041} C_VEL
LIN {X 0,Y 404.195,Z 667.945,A -85,B 0,C 180,E1 -10995.118,E2 -10995.118} C_VEL
LIN {X 0,Y 404.204,Z 667.938,A -85,B 0,C 180,E1 -10998.238,E2 -10998.238} C_VEL
LIN {X 0,Y 404.184,Z 667.945,A -85,B 0,C 180,E1 -11001.416,E2 -11001.416} C_VEL
LIN {X 0,Y 404.206,Z 667.944,A -85,B 0,C 180,E1 -11005.297,E2 -11005.297} C_VEL
LIN {X 0,Y 404.188,Z 667.909,A -85,B 0,C 180,E1 -11008,E2 -11008} C_VEL
LIN {X 0,Y 404.133,Z 667.953,A -85,B 0,C 180,E1 -11011.559,E2 -11011.559} C_VEL
LIN {X 0,Y 404.176,Z 667.923,A -85,B 0,C 180,E1 -11015.016,E2 -11015.016} C_VEL
LIN {X 0,Y 404.155,Z 667.95,A -85,B 0,C 180,E1 -11018.756,E2 -11018.756} C_VEL
LIN {X 0,Y 404.183,Z 667.952,A -85,B 0,C 180,E1 -11021.611,E2 -11021.611} C_VEL
LIN {X 0,Y 404.182,Z 667.951,A -85,B 0,C 180,E1 -11024.529,E2 -11024.529} C_VEL
LIN {X 0,Y 404.163,Z 667.954,A -85,B 0,C 180,E1 -11027.3,E2 -11027.3} C_VEL
LIN {X 0,Y 404.162,Z 667.953,A -85,B 0,C 180,E1 -11029.956,E2 -11029.956} C_VEL
LIN {X 0,Y 404.134,Z 667.957,A -85,B 0,C 180,E1 -11033.125,E2 -11033.125} C_VEL
LIN {X 0,Y 404.139,Z 667.958,A -85,B 0,C 180,E1 -11036.188,E2 -11036.188} C_VEL
LIN {X 0,Y 404.148,Z 667.956,A -85,B 0,C 180,E1 -11039.716,E2 -11039.716} C_VEL
LIN {X 0,Y 404.19,Z 667.951,A -85,B 0,C 180,E1 -11043.123,E2 -11043.123} C_VEL
LIN {X 0,Y 404.172,Z 667.952,A -85,B 0,C 180,E1 -11045.335,E2 -11045.335} C_VEL
LIN {X 0,Y 404.134,Z 667.959,A -85,B 0,C 180,E1 -11048.581,E2 -11048.581} C_VEL
LIN {X 0,Y 404.206,Z 667.948,A -85,B 0,C 180,E1 -11051.762,E2 -11051.762} C_VEL
LIN {X 0,Y 404.202,Z 667.949,A -85,B 0,C 180,E1 -11054.882,E2 -11054.882} C_VEL
LIN {X 0,Y 404.252,Z 667.944,A -85,B 0,C 180,E1 -11057.959,E2 -11057.959} C_VEL
LIN {X 0,Y 404.43,Z 667.923,A -85,B 0,C 180,E1 -11062.1,E2 -11062.1} C_VEL
LIN {X 0,Y 404.42,Z 667.921,A -85,B 0,C 180,E1 -11064.015,E2 -11064.015} C_VEL
LIN {X 0,Y 404.479,Z 667.914,A -85,B 0,C 180,E1 -11068.009,E2 -11068.009} C_VEL
LIN {X 0,Y 404.608,Z 667.901,A -85,B 0,C 180,E1 -11070,E2 -11070} C_VEL
LIN {X 0,Y 404.42,Z 667.922,A -85,B 0,C 180,E1 -11072.988,E2 -11072.988} C_VEL
LIN {X 0,Y 404.408,Z 667.923,A -85,B 0,C 180,E1 -11076.987,E2 -11076.987} C_VEL
LIN {X 0,Y 404.254,Z 667.942,A -85,B 0,C 180,E1 -11080.012,E2 -11080.012} C_VEL
LIN {X 0,Y 404.262,Z 667.943,A -85,B 0,C 180,E1 -11083.211,E2 -11083.211} C_VEL
LIN {X 0,Y 404.211,Z 667.947,A -85,B 0,C 180,E1 -11087.007,E2 -11087.007} C_VEL
LIN {X 0,Y 404.159,Z 667.954,A -85,B 0,C 180,E1 -11090.351,E2 -11090.351} C_VEL
LIN {X 0,Y 404.131,Z 667.958,A -85,B 0,C 180,E1 -11091.924,E2 -11091.924} C_VEL
LIN {X 0,Y 403.489,Z 668.039,A -85,B 0,C 180,E1 -11092.755,E2 -11092.755} C_VEL
LIN {X 0,Y 400.656,Z 668.396,A -85,B 0,C 180,E1 -11094.107,E2 -11094.107} C_VEL
LIN {X 0,Y 398.246,Z 668.696,A -85,B 0,C 180,E1 -11095.199,E2 -11095.199} C_VEL
LIN {X 0,Y 397.212,Z 668.821,A -85,B 0,C 180,E1 -11096.044,E2 -11096.044} C_VEL
LIN {X 0,Y 397.129,Z 668.83,A -85,B 0,C 180,E1 -11096.329,E2 -11096.329} C_VEL
LIN {X 0,Y 397.121,Z 668.831,A -85,B 0,C 180,E1 -11098.543,E2 -11098.543} C_VEL
LIN {X 0,Y 397.075,Z 668.838,A -85,B 0,C 180,E1 -11102.071,E2 -11102.071} C_VEL
LIN {X 0,Y 397.113,Z 668.831,A -85,B 0,C 180,E1 -11105.503,E2 -11105.503} C_VEL
LIN {X 0,Y 397.13,Z 668.831,A -85,B 0,C 180,E1 -11108.862,E2 -11108.862} C_VEL
LIN {X 0,Y 397.106,Z 668.834,A -85,B 0,C 180,E1 -11112.261,E2 -11112.261} C_VEL
LIN {X 0,Y 397.108,Z 668.835,A -85,B 0,C 180,E1 -11115.064,E2 -11115.064} C_VEL
LIN {X 0,Y 397.148,Z 668.827,A -85,B 0,C 180,E1 -11118.006,E2 -11118.006} C_VEL
LIN {X 0,Y 397.101,Z 668.824,A -85,B 0,C 180,E1 -11121.726,E2 -11121.726} C_VEL
LIN {X 0,Y 397.117,Z 668.81,A -85,B 0,C 180,E1 -11125.506,E2 -11125.506} C_VEL
LIN {X 0,Y 397.074,Z 668.818,A -85,B 0,C 180,E1 -11129.118,E2 -11129.118} C_VEL
LIN {X 0,Y 397.185,Z 668.789,A -85,B 0,C 180,E1 -11132.61,E2 -11132.61} C_VEL
LIN {X 0,Y 397.126,Z 668.828,A -85,B 0,C 180,E1 -11135.982,E2 -11135.982} C_VEL
LIN {X 0,Y 397.146,Z 668.823,A -85,B 0,C 180,E1 -11139.273,E2 -11139.273} C_VEL
LIN {X 0,Y 397.172,Z 668.812,A -85,B 0,C 180,E1 -11142.845,E2 -11142.845} C_VEL
LIN {X 0,Y 397.219,Z 668.8,A -85,B 0,C 180,E1 -11146.703,E2 -11146.703} C_VEL
LIN {X 0,Y 397.215,Z 668.816,A -85,B 0,C 180,E1 -11149.809,E2 -11149.809} C_VEL
LIN {X 0,Y 397.341,Z 668.791,A -85,B 0,C 180,E1 -11152.888,E2 -11152.888} C_VEL
LIN {X 0,Y 397.253,Z 668.812,A -85,B 0,C 180,E1 -11154.925,E2 -11154.925} C_VEL
LIN {X 0,Y 397.442,Z 668.773,A -85,B 0,C 180,E1 -11157.974,E2 -11157.974} C_VEL
LIN {X 0,Y 397.572,Z 668.772,A -85,B 0,C 180,E1 -11160,E2 -11160} C_VEL
LIN {X 0,Y 397.374,Z 668.785,A -85,B 0,C 180,E1 -11163.042,E2 -11163.042} C_VEL
LIN {X 0,Y 397.378,Z 668.794,A -85,B 0,C 180,E1 -11166.092,E2 -11166.092} C_VEL
LIN {X 0,Y 397.249,Z 668.804,A -85,B 0,C 180,E1 -11169.162,E2 -11169.162} C_VEL
LIN {X 0,Y 397.222,Z 668.807,A -85,B 0,C 180,E1 -11172.258,E2 -11172.258} C_VEL
LIN {X 0,Y 397.171,Z 668.825,A -85,B 0,C 180,E1 -11175.392,E2 -11175.392} C_VEL
LIN {X 0,Y 397.162,Z 668.814,A -85,B 0,C 180,E1 -11178.574,E2 -11178.574} C_VEL
LIN {X 0,Y 397.09,Z 668.822,A -85,B 0,C 180,E1 -11181.819,E2 -11181.819} C_VEL
LIN {X 0,Y 397.149,Z 668.827,A -85,B 0,C 180,E1 -11185.132,E2 -11185.132} C_VEL
LIN {X 0,Y 397.155,Z 668.783,A -85,B 0,C 180,E1 -11187.777,E2 -11187.777} C_VEL
LIN {X 0,Y 397.077,Z 668.818,A -85,B 0,C 180,E1 -11190.883,E2 -11190.883} C_VEL
LIN {X 0,Y 397.119,Z 668.812,A -85,B 0,C 180,E1 -11194.494,E2 -11194.494} C_VEL
LIN {X 0,Y 397.104,Z 668.833,A -85,B 0,C 180,E1 -11198.275,E2 -11198.275} C_VEL
LIN {X 0,Y 397.151,Z 668.807,A -85,B 0,C 180,E1 -11201.994,E2 -11201.994} C_VEL
LIN {X 0,Y 397.109,Z 668.813,A -85,B 0,C 180,E1 -11205.066,E2 -11205.066} C_VEL
LIN {X 0,Y 397.063,Z 668.831,A -85,B 0,C 180,E1 -11208.022,E2 -11208.022} C_VEL
LIN {X 0,Y 397.104,Z 668.978,A -85,B 0,C 180,E1 -11209.684,E2 -11209.684} C_VEL
LIN {X 0,Y 399.871,Z 678.963,A -85,B 0,C 180,E1 -11212.27,E2 -11212.27} C_VEL
LIN {X 0,Y 402.813,Z 690.144,A -85,B 0,C 180,E1 -11214.939,E2 -11214.939} C_VEL
LIN {X 0,Y 403.253,Z 691.526,A -85,B 0,C 180,E1 -11215.138,E2 -11215.138} C_VEL
LIN {X 0,Y 412.168,Z 710.074,A -85,B 0,C 180,E1 -11216.38,E2 -11216.38} C_VEL
LIN {X 0,Y 418.313,Z 736.15,A -85,B 0,C 180,E1 -11217.455,E2 -11217.455} C_VEL
LIN {X 0,Y 414.637,Z 893.739,A -85,B 0,C 180,E1 -11220.285,E2 -11220.285} C_VEL
LIN {X 0,Y 413.93,Z 906.655,A -85,B 0,C 180,E1 -11220.608,E2 -11220.608} C_VEL
LIN {X 0,Y 412.981,Z 919.011,A -85,B 0,C 180,E1 -11221.023,E2 -11221.023} C_VEL
LIN {X 0,Y 412.011,Z 932.136,A -85,B 0,C 180,E1 -11221.61,E2 -11221.61} C_VEL
LIN {X 0,Y 410.865,Z 943.523,A -85,B 0,C 180,E1 -11222.218,E2 -11222.218} C_VEL
LIN {X 0,Y 409.533,Z 955.756,A -85,B 0,C 180,E1 -11223.006,E2 -11223.006} C_VEL
LIN {X 0,Y 408.07,Z 968.137,A -85,B 0,C 180,E1 -11223.956,E2 -11223.956} C_VEL
LIN {X 0,Y 406.382,Z 980.502,A -85,B 0,C 180,E1 -11225.069,E2 -11225.069} C_VEL
LIN {X 0,Y 404.916,Z 991.306,A -85,B 0,C 180,E1 -11226.201,E2 -11226.201} C_VEL
LIN {X 0,Y 403.397,Z 1001.808,A -85,B 0,C 180,E1 -11227.463,E2 -11227.463} C_VEL
LIN {X 0,Y 402.003,Z 1011.079,A -85,B 0,C 180,E1 -11228.731,E2 -11228.731} C_VEL
LIN {X 0,Y 400.63,Z 1020.816,A -85,B 0,C 180,E1 -11230.264,E2 -11230.264} C_VEL
LIN {X 0,Y 399.308,Z 1030.396,A -85,B 0,C 180,E1 -11232.014,E2 -11232.014} C_VEL
LIN {X 0,Y 398.354,Z 1037.946,A -85,B 0,C 180,E1 -11233.604,E2 -11233.604} C_VEL
LIN {X 0,Y 397.561,Z 1044.376,A -85,B 0,C 180,E1 -11235.148,E2 -11235.148} C_VEL
LIN {X 0,Y 396.815,Z 1051.915,A -85,B 0,C 180,E1 -11237.299,E2 -11237.299} C_VEL
LIN {X 0,Y 396.408,Z 1056.287,A -85,B 0,C 180,E1 -11238.754,E2 -11238.754} C_VEL
LIN {X 0,Y 396.023,Z 1061.38,A -85,B 0,C 180,E1 -11240.81,E2 -11240.81} C_VEL
LIN {X 0,Y 395.89,Z 1065.375,A -85,B 0,C 180,E1 -11242.862,E2 -11242.862} C_VEL
LIN {X 0,Y 395.839,Z 1067.046,A -85,B 0,C 180,E1 -11243.885,E2 -11243.885} C_VEL
LIN {X 0,Y 395.733,Z 1069.506,A -85,B 0,C 180,E1 -11245.927,E2 -11245.927} C_VEL
LIN {X 0,Y 395.751,Z 1070.97,A -85,B 0,C 180,E1 -11247.965,E2 -11247.965} C_VEL
LIN {X 0,Y 395.774,Z 1071.456,A -85,B 0,C 180,E1 -11250,E2 -11250} C_VEL
LIN {X 0,Y 395.751,Z 1070.97,A -85,B 0,C 180,E1 -11252.035,E2 -11252.035} C_VEL
LIN {X 0,Y 395.733,Z 1069.506,A -85,B 0,C 180,E1 -11254.073,E2 -11254.073} C_VEL
LIN {X 0,Y 395.857,Z 1066.962,A -85,B 0,C 180,E1 -11256.166,E2 -11256.166} C_VEL
LIN {X 0,Y 395.988,Z 1062.467,A -85,B 0,C 180,E1 -11258.676,E2 -11258.676} C_VEL
LIN {X 0,Y 396.129,Z 1058.98,A -85,B 0,C 180,E1 -11260.219,E2 -11260.219} C_VEL
LIN {X 0,Y 396.67,Z 1053.259,A -85,B 0,C 180,E1 -11262.275,E2 -11262.275} C_VEL
LIN {X 0,Y 397.158,Z 1048.199,A -85,B 0,C 180,E1 -11263.821,E2 -11263.821} C_VEL
LIN {X 0,Y 398.038,Z 1040.167,A -85,B 0,C 180,E1 -11265.883,E2 -11265.883} C_VEL
LIN {X 0,Y 399.004,Z 1033.185,A -85,B 0,C 180,E1 -11267.423,E2 -11267.423} C_VEL
LIN {X 0,Y 399.998,Z 1025.212,A -85,B 0,C 180,E1 -11268.968,E2 -11268.968} C_VEL
LIN {X 0,Y 401.32,Z 1016.098,A -85,B 0,C 180,E1 -11270.502,E2 -11270.502} C_VEL
LIN {X 0,Y 402.592,Z 1007.551,A -85,B 0,C 180,E1 -11271.771,E2 -11271.771} C_VEL
LIN {X 0,Y 404.245,Z 995.66,A -85,B 0,C 180,E1 -11273.297,E2 -11273.297} C_VEL
LIN {X 0,Y 405.901,Z 984.244,A -85,B 0,C 180,E1 -11274.553,E2 -11274.553} C_VEL
LIN {X 0,Y 407.23,Z 973.816,A -85,B 0,C 180,E1 -11275.559,E2 -11275.559} C_VEL
LIN {X 0,Y 408.824,Z 961.79,A -85,B 0,C 180,E1 -11276.548,E2 -11276.548} C_VEL
LIN {X 0,Y 410.206,Z 949.665,A -85,B 0,C 180,E1 -11277.401,E2 -11277.401} C_VEL
LIN {X 0,Y 411.538,Z 936.921,A -85,B 0,C 180,E1 -11278.148,E2 -11278.148} C_VEL
LIN {X 0,Y 412.667,Z 923.49,A -85,B 0,C 180,E1 -11278.792,E2 -11278.792} C_VEL
LIN {X 0,Y 413.639,Z 910.571,A -85,B 0,C 180,E1 -11279.275,E2 -11279.275} C_VEL
LIN {X 0,Y 414.507,Z 897.424,A -85,B 0,C 180,E1 -11279.634,E2 -11279.634} C_VEL
LIN {X 0,Y 415.221,Z 872.271,A -85,B 0,C 180,E1 -11280.118,E2 -11280.118} C_VEL
LIN {X 0,Y 418.321,Z 736.04,A -85,B 0,C 180,E1 -11282.547,E2 -11282.547} C_VEL
LIN {X 0,Y 412.205,Z 710.183,A -85,B 0,C 180,E1 -11283.614,E2 -11283.614} C_VEL
LIN {X 0,Y 403.107,Z 690.994,A -85,B 0,C 180,E1 -11284.902,E2 -11284.902} C_VEL
LIN {X 0,Y 400.507,Z 681.342,A -85,B 0,C 180,E1 -11287.145,E2 -11287.145} C_VEL
LIN {X 0,Y 397.214,Z 669.411,A -85,B 0,C 180,E1 -11290.152,E2 -11290.152} C_VEL
LIN {X 0,Y 397.097,Z 668.833,A -85,B 0,C 180,E1 -11290.445,E2 -11290.445} C_VEL
LIN {X 0,Y 397.1,Z 668.818,A -85,B 0,C 180,E1 -11293.647,E2 -11293.647} C_VEL
LIN {X 0,Y 397.159,Z 668.826,A -85,B 0,C 180,E1 -11296.511,E2 -11296.511} C_VEL
LIN {X 0,Y 397.118,Z 668.81,A -85,B 0,C 180,E1 -11299.55,E2 -11299.55} C_VEL
LIN {X 0,Y 397.093,Z 668.82,A -85,B 0,C 180,E1 -11302.789,E2 -11302.789} C_VEL
LIN {X 0,Y 397.111,Z 668.825,A -85,B 0,C 180,E1 -11306.281,E2 -11306.281} C_VEL
LIN {X 0,Y 397.106,Z 668.791,A -85,B 0,C 180,E1 -11310.133,E2 -11310.133} C_VEL
LIN {X 0,Y 397.187,Z 668.786,A -85,B 0,C 180,E1 -11312.609,E2 -11312.609} C_VEL
LIN {X 0,Y 397.125,Z 668.831,A -85,B 0,C 180,E1 -11315.981,E2 -11315.981} C_VEL
LIN {X 0,Y 397.146,Z 668.825,A -85,B 0,C 180,E1 -11319.698,E2 -11319.698} C_VEL
LIN {X 0,Y 397.173,Z 668.815,A -85,B 0,C 180,E1 -11322.844,E2 -11322.844} C_VEL
LIN {X 0,Y 397.218,Z 668.806,A -85,B 0,C 180,E1 -11326.678,E2 -11326.678} C_VEL
LIN {X 0,Y 397.221,Z 668.814,A -85,B 0,C 180,E1 -11329.809,E2 -11329.809} C_VEL
LIN {X 0,Y 397.348,Z 668.787,A -85,B 0,C 180,E1 -11332.888,E2 -11332.888} C_VEL
LIN {X 0,Y 397.253,Z 668.814,A -85,B 0,C 180,E1 -11334.925,E2 -11334.925} C_VEL
LIN {X 0,Y 397.442,Z 668.78,A -85,B 0,C 180,E1 -11337.973,E2 -11337.973} C_VEL
LIN {X 0,Y 397.572,Z 668.771,A -85,B 0,C 180,E1 -11340,E2 -11340} C_VEL
LIN {X 0,Y 397.374,Z 668.782,A -85,B 0,C 180,E1 -11343.041,E2 -11343.041} C_VEL
LIN {X 0,Y 397.344,Z 668.793,A -85,B 0,C 180,E1 -11346.587,E2 -11346.587} C_VEL
LIN {X 0,Y 397.247,Z 668.807,A -85,B 0,C 180,E1 -11349.162,E2 -11349.162} C_VEL
LIN {X 0,Y 397.21,Z 668.803,A -85,B 0,C 180,E1 -11352.258,E2 -11352.258} C_VEL
LIN {X 0,Y 397.169,Z 668.822,A -85,B 0,C 180,E1 -11355.392,E2 -11355.392} C_VEL
LIN {X 0,Y 397.162,Z 668.818,A -85,B 0,C 180,E1 -11358.573,E2 -11358.573} C_VEL
LIN {X 0,Y 397.15,Z 668.818,A -85,B 0,C 180,E1 -11361.815,E2 -11361.815} C_VEL
LIN {X 0,Y 397.143,Z 668.824,A -85,B 0,C 180,E1 -11365.513,E2 -11365.513} C_VEL
LIN {X 0,Y 397.116,Z 668.785,A -85,B 0,C 180,E1 -11368.544,E2 -11368.544} C_VEL
LIN {X 0,Y 397.071,Z 668.834,A -85,B 0,C 180,E1 -11372.072,E2 -11372.072} C_VEL
LIN {X 0,Y 397.111,Z 668.795,A -85,B 0,C 180,E1 -11375.504,E2 -11375.504} C_VEL
LIN {X 0,Y 397.129,Z 668.827,A -85,B 0,C 180,E1 -11378.863,E2 -11378.863} C_VEL
LIN {X 0,Y 397.152,Z 668.827,A -85,B 0,C 180,E1 -11382.256,E2 -11382.256} C_VEL
LIN {X 0,Y 397.103,Z 668.835,A -85,B 0,C 180,E1 -11385.066,E2 -11385.066} C_VEL
LIN {X 0,Y 397.102,Z 668.833,A -85,B 0,C 180,E1 -11388.015,E2 -11388.015} C_VEL
LIN {X 0,Y 397.13,Z 668.831,A -85,B 0,C 180,E1 -11391.138,E2 -11391.138} C_VEL
LIN {X 0,Y 397.113,Z 668.831,A -85,B 0,C 180,E1 -11394.497,E2 -11394.497} C_VEL
LIN {X 0,Y 397.075,Z 668.838,A -85,B 0,C 180,E1 -11397.929,E2 -11397.929} C_VEL
LIN {X 0,Y 397.121,Z 668.83,A -85,B 0,C 180,E1 -11401.457,E2 -11401.457} C_VEL
LIN {X 0,Y 397.148,Z 668.83,A -85,B 0,C 180,E1 -11404.488,E2 -11404.488} C_VEL
LIN {X 0,Y 397.104,Z 668.834,A -85,B 0,C 180,E1 -11407.086,E2 -11407.086} C_VEL
LIN {X 0,Y 397.143,Z 668.828,A -85,B 0,C 180,E1 -11410.353,E2 -11410.353} C_VEL
LIN {X 0,Y 397.162,Z 668.825,A -85,B 0,C 180,E1 -11413.553,E2 -11413.553} C_VEL
